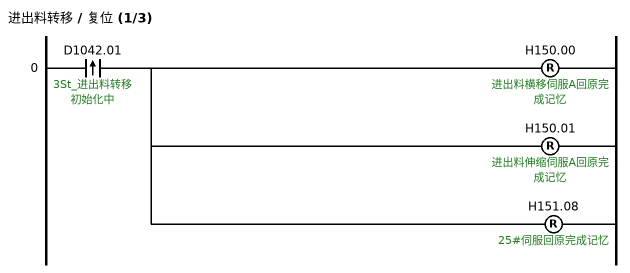
; rung 0
@LD D1042.01  ; 3St_进出料转移 初始化中
RSET H150.00  ; 进出料横移伺服A回原完成记忆
RSET H150.01  ; 进出料伸缩伺服A回原完成记忆
RSET H151.08  ; 25#伺服回原完成记忆

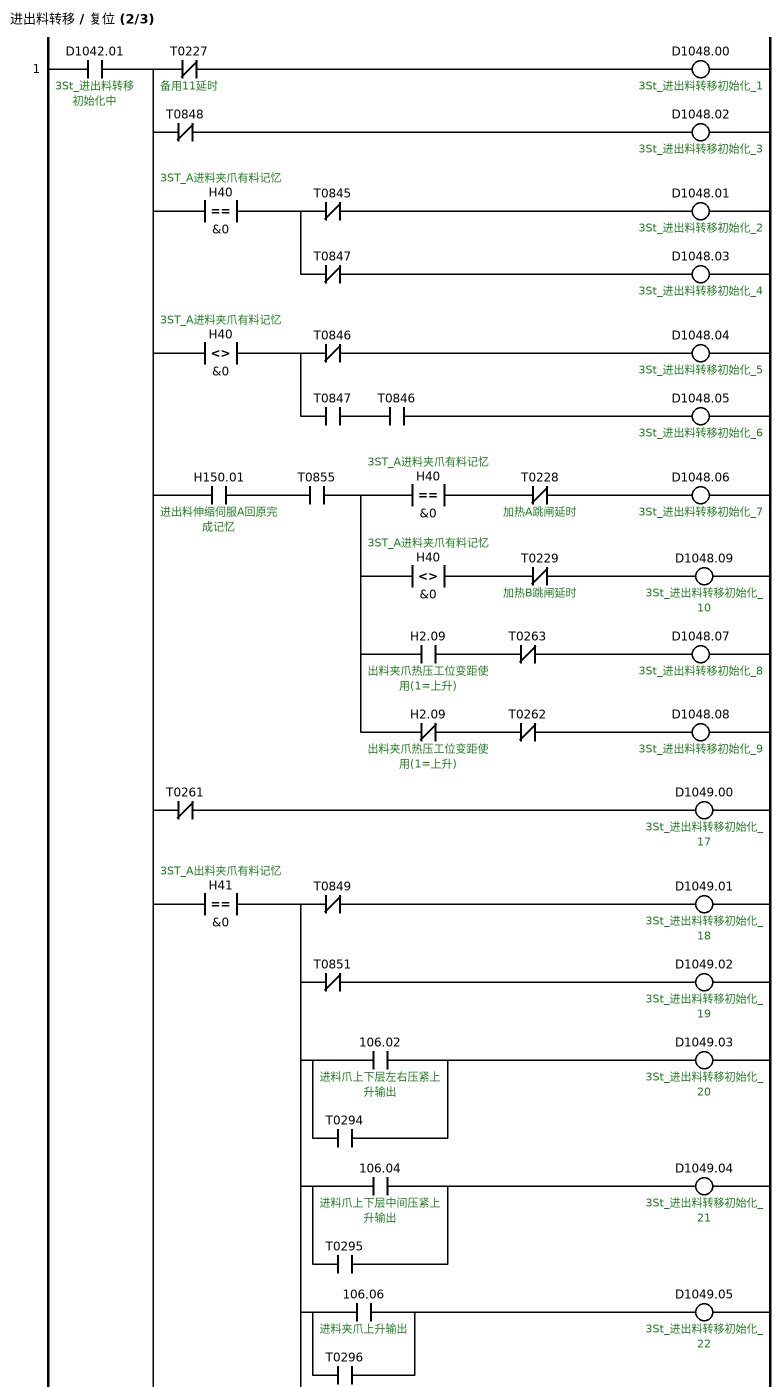

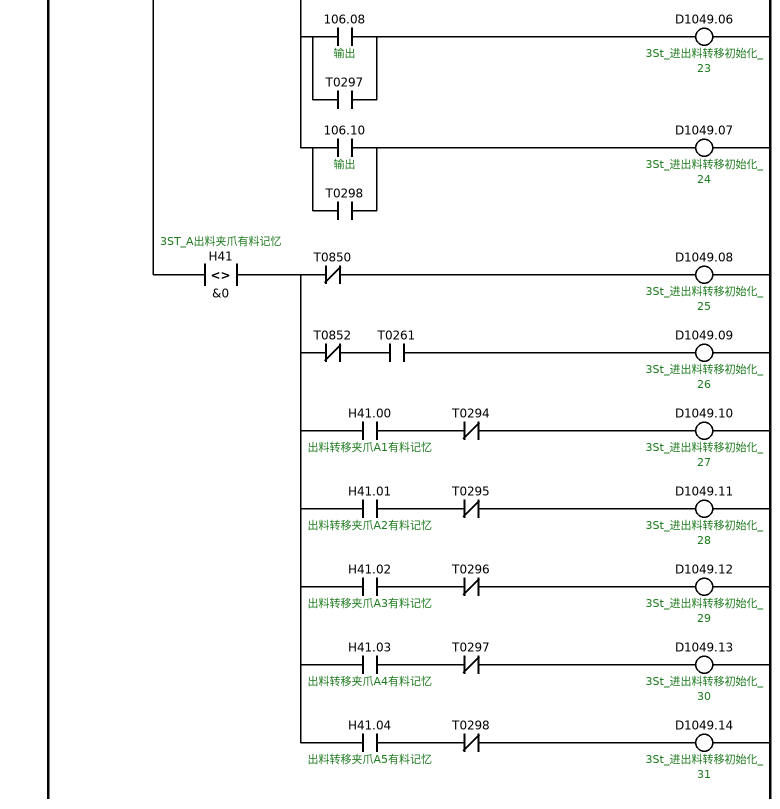
; rung 1
LD D1042.01  ; 3St_进出料转移 初始化中
OUT TR0
ANDNOT T0227  ; 备用11延时
OUT D1048.00  ; 3St_进出料转移初始化_1
LD TR0
ANDNOT T0848
OUT D1048.02  ; 3St_进出料转移初始化_3
LD TR0
AND=(300) H40 &0  ; 3ST_A进料夹爪有料记忆
OUT TR1
ANDNOT T0845
OUT D1048.01  ; 3St_进出料转移初始化_2
LD TR1
ANDNOT T0847
OUT D1048.03  ; 3St_进出料转移初始化_4
LD TR0
AND<>(305) H40 &0  ; 3ST_A进料夹爪有料记忆
OUT TR1
ANDNOT T0846
OUT D1048.04  ; 3St_进出料转移初始化_5
LD TR1
AND T0847
AND T0846
OUT D1048.05  ; 3St_进出料转移初始化_6
LD TR0
AND H150.01  ; 进出料伸缩伺服A回原完成记忆
AND T0855
OUT TR1
AND=(300) H40 &0  ; 3ST_A进料夹爪有料记忆
ANDNOT T0228  ; 加热A跳闸延时
OUT D1048.06  ; 3St_进出料转移初始化_7
LD TR1
AND<>(305) H40 &0  ; 3ST_A进料夹爪有料记忆
ANDNOT T0229  ; 加热B跳闸延时
OUT D1048.09  ; 3St_进出料转移初始化_10
LD TR1
AND H2.09  ; 出料夹爪热压工位变距使用(1=上升)
ANDNOT T0263
OUT D1048.07  ; 3St_进出料转移初始化_8
LD TR1
ANDNOT H2.09  ; 出料夹爪热压工位变距使用(1=上升)
ANDNOT T0262
OUT D1048.08  ; 3St_进出料转移初始化_9
LD TR0
ANDNOT T0261
OUT D1049.00  ; 3St_进出料转移初始化_17
LD TR0
AND=(300) H41 &0  ; 3ST_A出料夹爪有料记忆
OUT TR1
ANDNOT T0849
OUT D1049.01  ; 3St_进出料转移初始化_18
LD TR1
ANDNOT T0851
OUT D1049.02  ; 3St_进出料转移初始化_19
LD TR1
LD 106.02  ; 进料爪上下层左右压紧上升输出
OR T0294
ANDLD
OUT D1049.03  ; 3St_进出料转移初始化_20
LD TR1
LD 106.04  ; 进料爪上下层中间压紧上升输出
OR T0295
ANDLD
OUT D1049.04  ; 3St_进出料转移初始化_21
LD TR1
LD 106.06  ; 进料夹爪上升输出
OR T0296
ANDLD
OUT D1049.05  ; 3St_进出料转移初始化_22
LD TR1
LD 106.08  ; 输出
OR T0297
ANDLD
OUT D1049.06  ; 3St_进出料转移初始化_23
LD TR1
LD 106.10  ; 输出
OR T0298
ANDLD
OUT D1049.07  ; 3St_进出料转移初始化_24
LD TR0
AND<>(305) H41 &0  ; 3ST_A出料夹爪有料记忆
OUT TR0
ANDNOT T0850
OUT D1049.08  ; 3St_进出料转移初始化_25
LD TR0
ANDNOT T0852
AND T0261
OUT D1049.09  ; 3St_进出料转移初始化_26
LD TR0
AND H41.00  ; 出料转移夹爪A1有料记忆
ANDNOT T0294
OUT D1049.10  ; 3St_进出料转移初始化_27
LD TR0
AND H41.01  ; 出料转移夹爪A2有料记忆
ANDNOT T0295
OUT D1049.11  ; 3St_进出料转移初始化_28
LD TR0
AND H41.02  ; 出料转移夹爪A3有料记忆
ANDNOT T0296
OUT D1049.12  ; 3St_进出料转移初始化_29
LD TR0
AND H41.03  ; 出料转移夹爪A4有料记忆
ANDNOT T0297
OUT D1049.13  ; 3St_进出料转移初始化_30
LD TR0
AND H41.04  ; 出料转移夹爪A5有料记忆
ANDNOT T0298
OUT D1049.14  ; 3St_进出料转移初始化_31

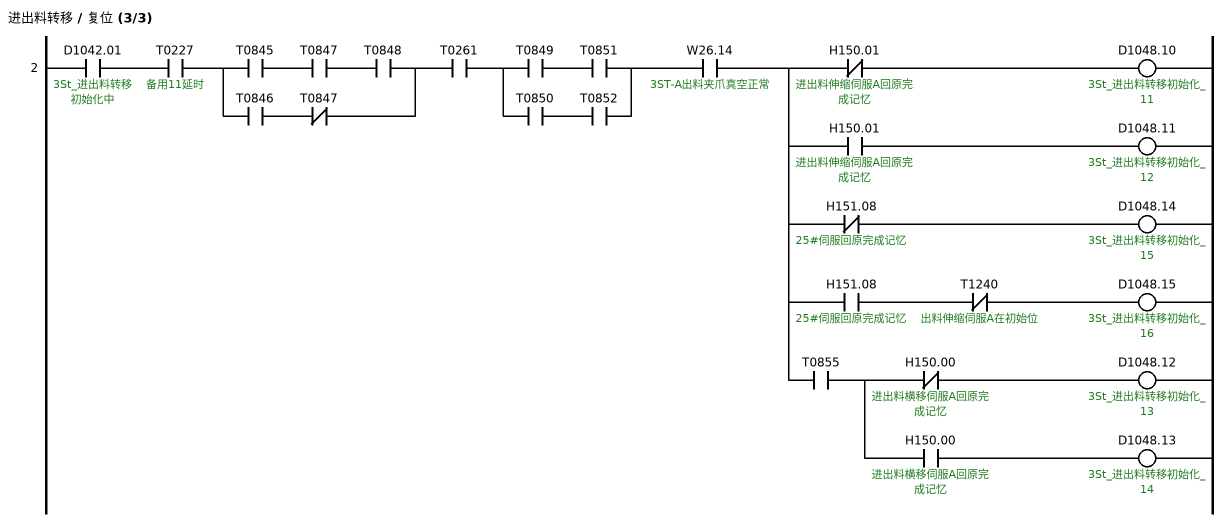
; rung 2
LD D1042.01  ; 3St_进出料转移 初始化中
AND T0227  ; 备用11延时
LD T0845
AND T0847
AND T0848
LD T0846
ANDNOT T0847
ORLD
ANDLD
AND T0261
LD T0849
AND T0851
LD T0850
AND T0852
ORLD
ANDLD
AND W26.14  ; 3ST-A出料夹爪真空正常
OUT TR0
ANDNOT H150.01  ; 进出料伸缩伺服A回原完成记忆
OUT D1048.10  ; 3St_进出料转移初始化_11
LD TR0
AND H150.01  ; 进出料伸缩伺服A回原完成记忆
OUT D1048.11  ; 3St_进出料转移初始化_12
LD TR0
ANDNOT H151.08  ; 25#伺服回原完成记忆
OUT D1048.14  ; 3St_进出料转移初始化_15
LD TR0
AND H151.08  ; 25#伺服回原完成记忆
ANDNOT T1240  ; 出料伸缩伺服A在初始位
OUT D1048.15  ; 3St_进出料转移初始化_16
LD TR0
AND T0855
OUT TR0
ANDNOT H150.00  ; 进出料横移伺服A回原完成记忆
OUT D1048.12  ; 3St_进出料转移初始化_13
LD TR0
AND H150.00  ; 进出料横移伺服A回原完成记忆
OUT D1048.13  ; 3St_进出料转移初始化_14

### Section 输出

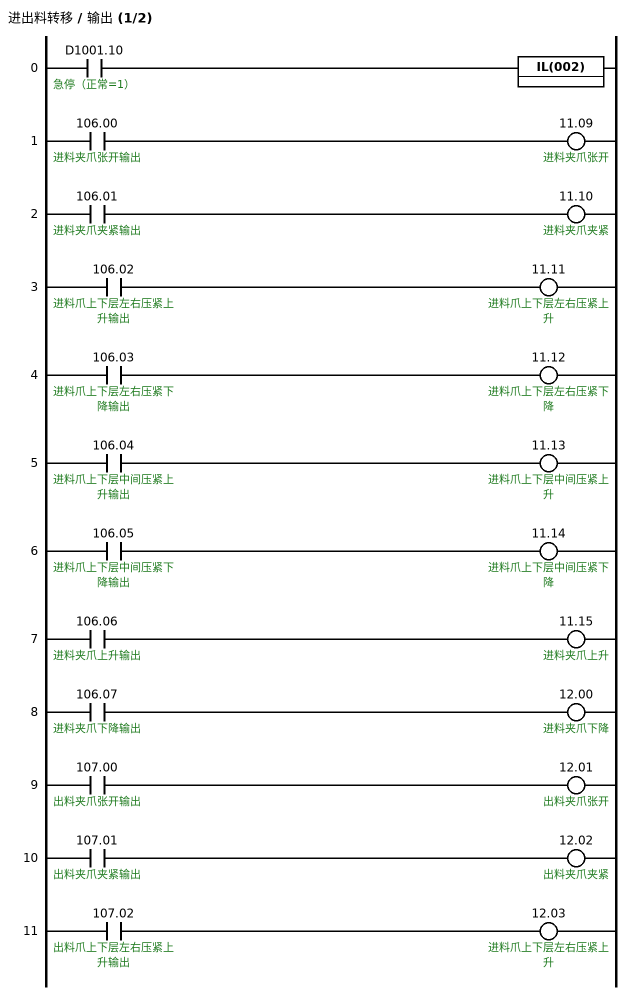
; rung 0
LD D1001.10  ; 急停（正常=1）
IL(002)
; rung 1
LD 106.00  ; 进料夹爪张开输出
OUT 11.09  ; 进料夹爪张开
; rung 2
LD 106.01  ; 进料夹爪夹紧输出
OUT 11.10  ; 进料夹爪夹紧
; rung 3
LD 106.02  ; 进料爪上下层左右压紧上升输出
OUT 11.11  ; 进料爪上下层左右压紧上升
; rung 4
LD 106.03  ; 进料爪上下层左右压紧下降输出
OUT 11.12  ; 进料爪上下层左右压紧下降
; rung 5
LD 106.04  ; 进料爪上下层中间压紧上升输出
OUT 11.13  ; 进料爪上下层中间压紧上升
; rung 6
LD 106.05  ; 进料爪上下层中间压紧下降输出
OUT 11.14  ; 进料爪上下层中间压紧下降
; rung 7
LD 106.06  ; 进料夹爪上升输出
OUT 11.15  ; 进料夹爪上升
; rung 8
LD 106.07  ; 进料夹爪下降输出
OUT 12.00  ; 进料夹爪下降
; rung 9
LD 107.00  ; 出料夹爪张开输出
OUT 12.01  ; 出料夹爪张开
; rung 10
LD 107.01  ; 出料夹爪夹紧输出
OUT 12.02  ; 出料夹爪夹紧
; rung 11
LD 107.02  ; 出料爪上下层左右压紧上升输出
OUT 12.03  ; 进料爪上下层左右压紧上升

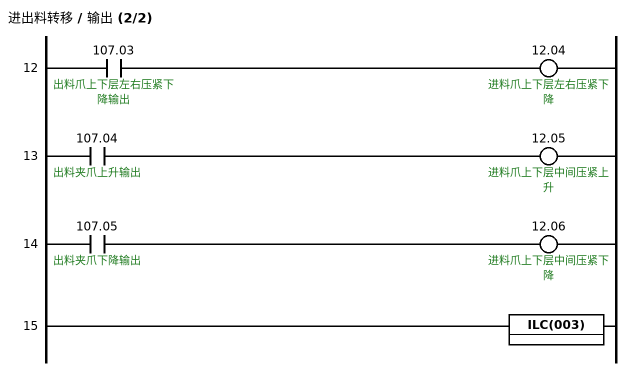
; rung 12
LD 107.03  ; 出料爪上下层左右压紧下降输出
OUT 12.04  ; 进料爪上下层左右压紧下降
; rung 13
LD 107.04  ; 出料夹爪上升输出
OUT 12.05  ; 进料爪上下层中间压紧上升
; rung 14
LD 107.05  ; 出料夹爪下降输出
OUT 12.06  ; 进料爪上下层中间压紧下降
; rung 15
ILC(003)

### Section END
; rung 0
END(001)

## Program 热压A (cyclic task 4)

### Section Main

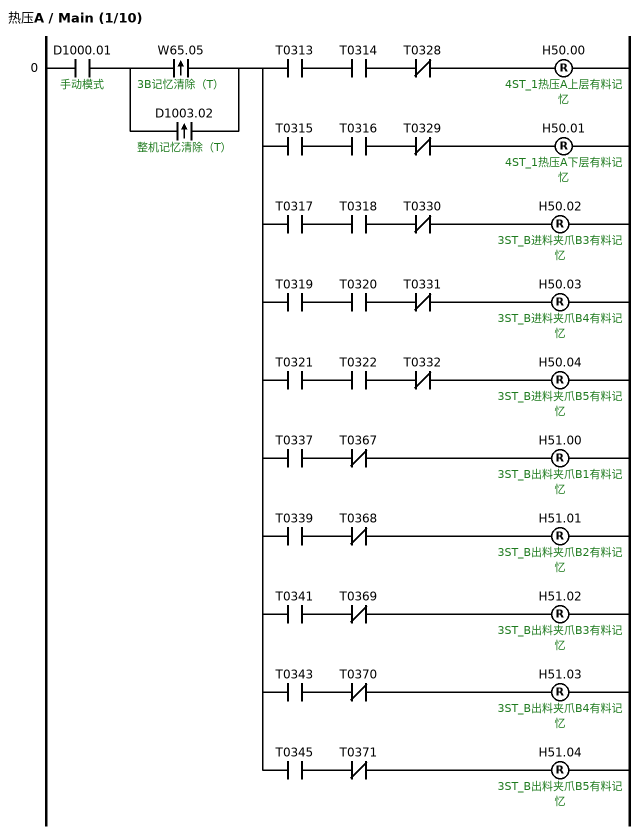
; rung 0
LD D1000.01  ; 手动模式
@LD W65.05  ; 3B记忆清除（T）
@OR D1003.02  ; 整机记忆清除（T）
ANDLD
OUT TR0
AND T0313
AND T0314
ANDNOT T0328
RSET H50.00  ; 4ST_1热压A上层有料记忆
LD TR0
AND T0315
AND T0316
ANDNOT T0329
RSET H50.01  ; 4ST_1热压A下层有料记忆
LD TR0
AND T0317
AND T0318
ANDNOT T0330
RSET H50.02  ; 3ST_B进料夹爪B3有料记忆
LD TR0
AND T0319
AND T0320
ANDNOT T0331
RSET H50.03  ; 3ST_B进料夹爪B4有料记忆
LD TR0
AND T0321
AND T0322
ANDNOT T0332
RSET H50.04  ; 3ST_B进料夹爪B5有料记忆
LD TR0
AND T0337
ANDNOT T0367
RSET H51.00  ; 3ST_B出料夹爪B1有料记忆
LD TR0
AND T0339
ANDNOT T0368
RSET H51.01  ; 3ST_B出料夹爪B2有料记忆
LD TR0
AND T0341
ANDNOT T0369
RSET H51.02  ; 3ST_B出料夹爪B3有料记忆
LD TR0
AND T0343
ANDNOT T0370
RSET H51.03  ; 3ST_B出料夹爪B4有料记忆
LD TR0
AND T0345
ANDNOT T0371
RSET H51.04  ; 3ST_B出料夹爪B5有料记忆

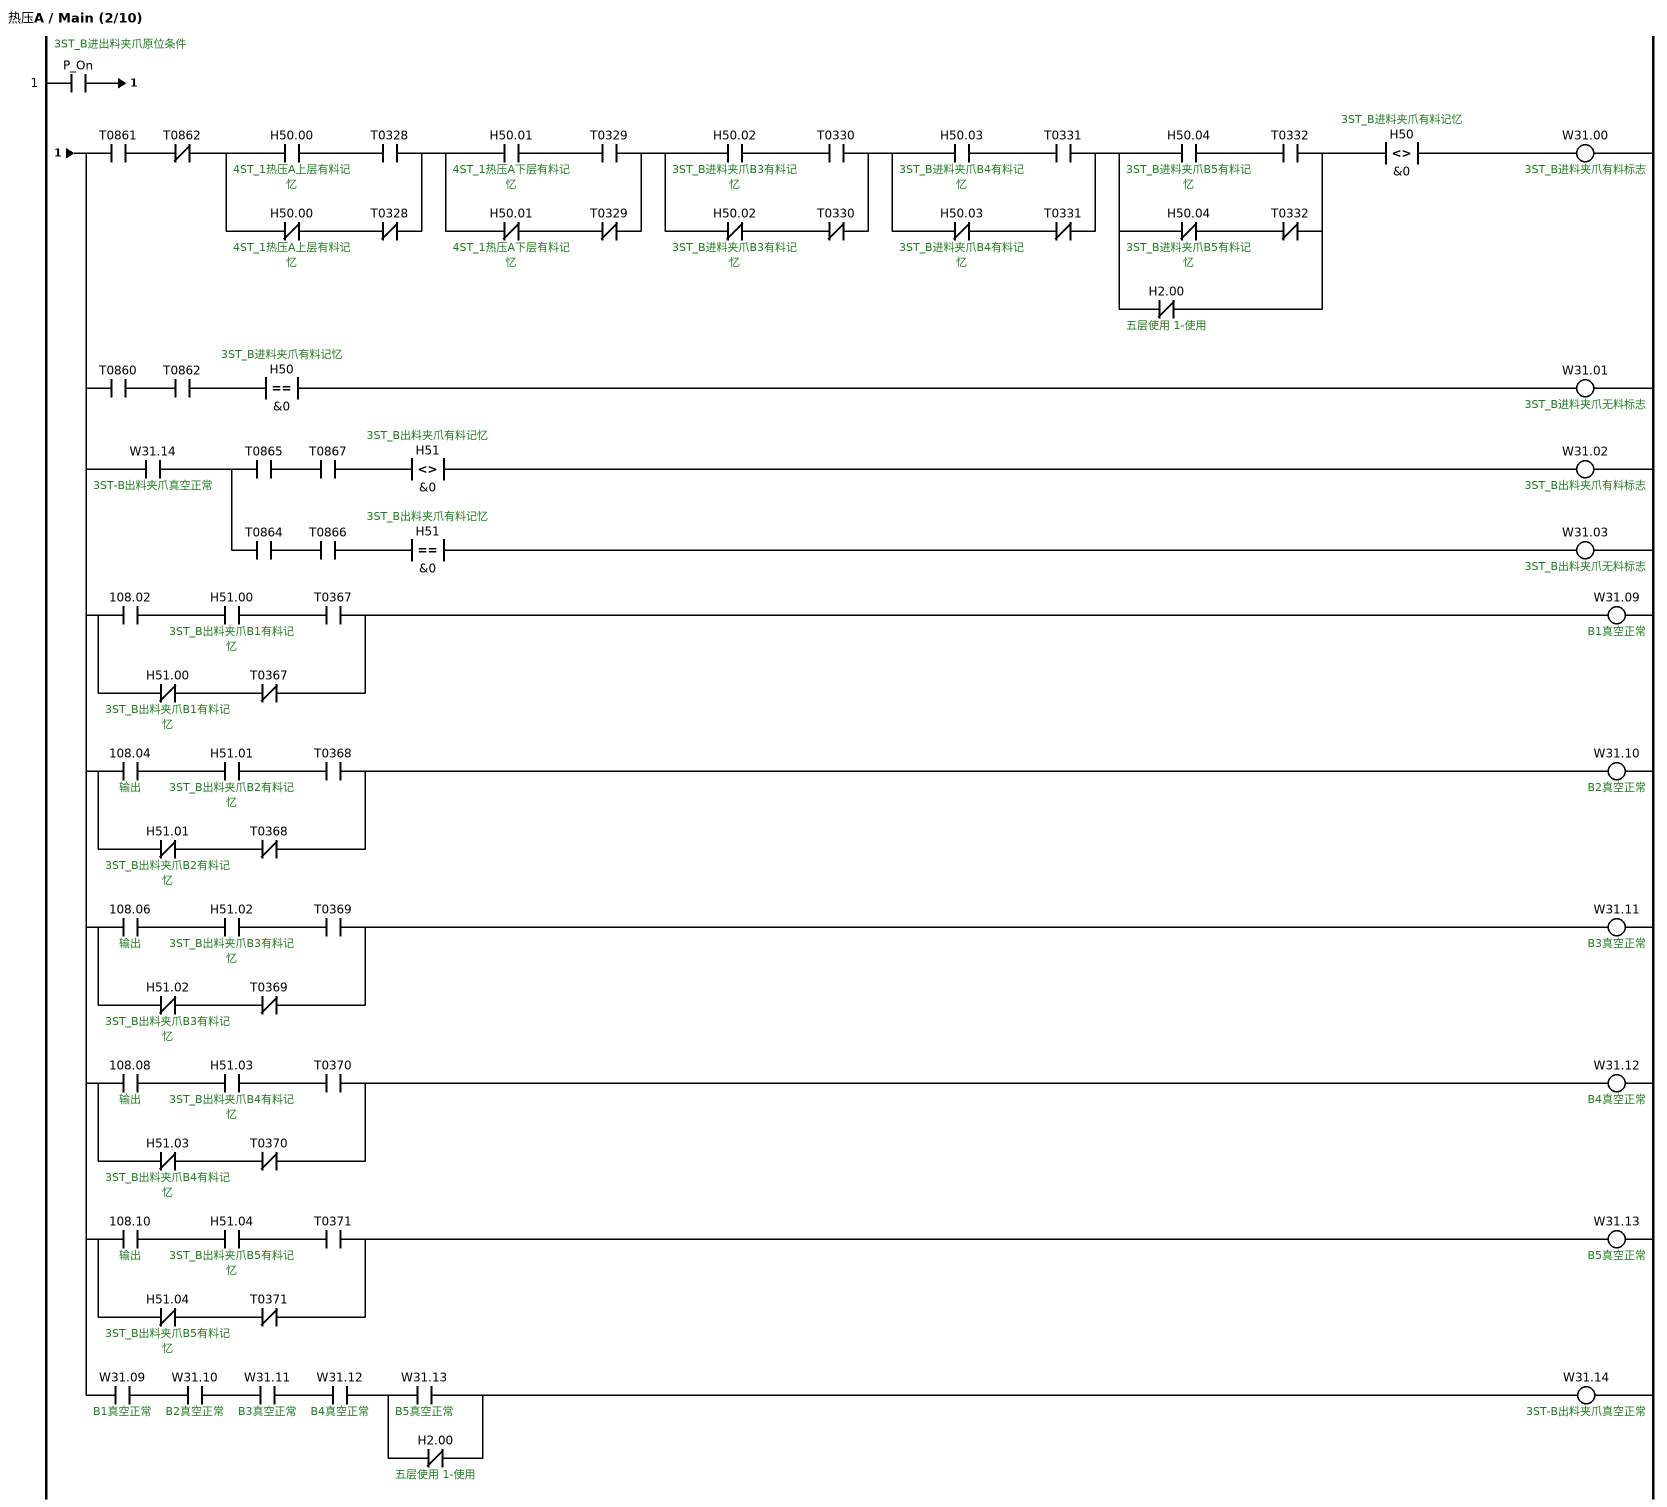
; rung 1: 3ST_B进出料夹爪原位条件
LD P_On
OUT TR0
AND T0861
ANDNOT T0862
LD H50.00  ; 4ST_1热压A上层有料记忆
AND T0328
LDNOT H50.00  ; 4ST_1热压A上层有料记忆
ANDNOT T0328
ORLD
ANDLD
LD H50.01  ; 4ST_1热压A下层有料记忆
AND T0329
LDNOT H50.01  ; 4ST_1热压A下层有料记忆
ANDNOT T0329
ORLD
ANDLD
LD H50.02  ; 3ST_B进料夹爪B3有料记忆
AND T0330
LDNOT H50.02  ; 3ST_B进料夹爪B3有料记忆
ANDNOT T0330
ORLD
ANDLD
LD H50.03  ; 3ST_B进料夹爪B4有料记忆
AND T0331
LDNOT H50.03  ; 3ST_B进料夹爪B4有料记忆
ANDNOT T0331
ORLD
ANDLD
LD H50.04  ; 3ST_B进料夹爪B5有料记忆
AND T0332
LDNOT H50.04  ; 3ST_B进料夹爪B5有料记忆
ANDNOT T0332
ORLD
ORNOT H2.00  ; 五层使用 1-使用
ANDLD
AND<>(305) H50 &0  ; 3ST_B进料夹爪有料记忆
OUT W31.00  ; 3ST_B进料夹爪有料标志
LD TR0
AND T0860
AND T0862
AND=(300) H50 &0  ; 3ST_B进料夹爪有料记忆
OUT W31.01  ; 3ST_B进料夹爪无料标志
LD TR0
AND W31.14  ; 3ST-B出料夹爪真空正常
OUT TR1
AND T0865
AND T0867
AND<>(305) H51 &0  ; 3ST_B出料夹爪有料记忆
OUT W31.02  ; 3ST_B出料夹爪有料标志
LD TR1
AND T0864
AND T0866
AND=(300) H51 &0  ; 3ST_B出料夹爪有料记忆
OUT W31.03  ; 3ST_B出料夹爪无料标志
LD TR0
LD 108.02
AND H51.00  ; 3ST_B出料夹爪B1有料记忆
AND T0367
LDNOT H51.00  ; 3ST_B出料夹爪B1有料记忆
ANDNOT T0367
ORLD
ANDLD
OUT W31.09  ; B1真空正常
LD TR0
LD 108.04  ; 输出
AND H51.01  ; 3ST_B出料夹爪B2有料记忆
AND T0368
LDNOT H51.01  ; 3ST_B出料夹爪B2有料记忆
ANDNOT T0368
ORLD
ANDLD
OUT W31.10  ; B2真空正常
LD TR0
LD 108.06  ; 输出
AND H51.02  ; 3ST_B出料夹爪B3有料记忆
AND T0369
LDNOT H51.02  ; 3ST_B出料夹爪B3有料记忆
ANDNOT T0369
ORLD
ANDLD
OUT W31.11  ; B3真空正常
LD TR0
LD 108.08  ; 输出
AND H51.03  ; 3ST_B出料夹爪B4有料记忆
AND T0370
LDNOT H51.03  ; 3ST_B出料夹爪B4有料记忆
ANDNOT T0370
ORLD
ANDLD
OUT W31.12  ; B4真空正常
LD TR0
LD 108.10  ; 输出
AND H51.04  ; 3ST_B出料夹爪B5有料记忆
AND T0371
LDNOT H51.04  ; 3ST_B出料夹爪B5有料记忆
ANDNOT T0371
ORLD
ANDLD
OUT W31.13  ; B5真空正常
LD TR0
AND W31.09  ; B1真空正常
AND W31.10  ; B2真空正常
AND W31.11  ; B3真空正常
AND W31.12  ; B4真空正常
LD W31.13  ; B5真空正常
ORNOT H2.00  ; 五层使用 1-使用
ANDLD
OUT W31.14  ; 3ST-B出料夹爪真空正常

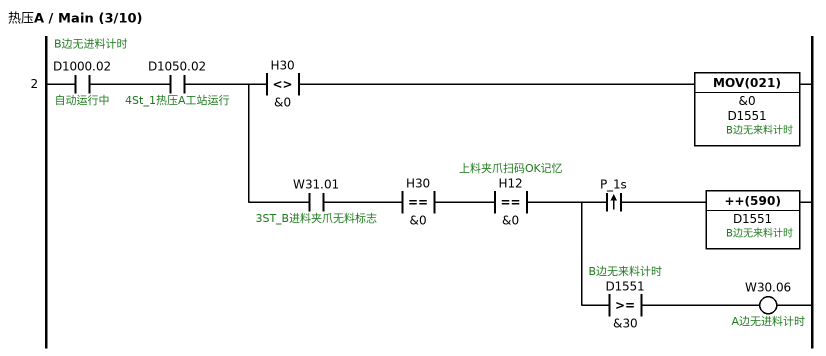
; rung 2: B边无进料计时
LD D1000.02  ; 自动运行中
AND D1050.02  ; 4St_1热压A工站运行
OUT TR0
AND<>(305) H30 &0
MOV(021) &0 D1551  ; B边无来料计时
LD TR0
AND W31.01  ; 3ST_B进料夹爪无料标志
AND=(300) H30 &0
AND=(300) H12 &0  ; 上料夹爪扫码OK记忆
OUT TR0
@AND P_1s
++(590) D1551  ; B边无来料计时
LD TR0
AND>=(325) D1551 &30  ; B边无来料计时
OUT W30.06  ; A边无进料计时

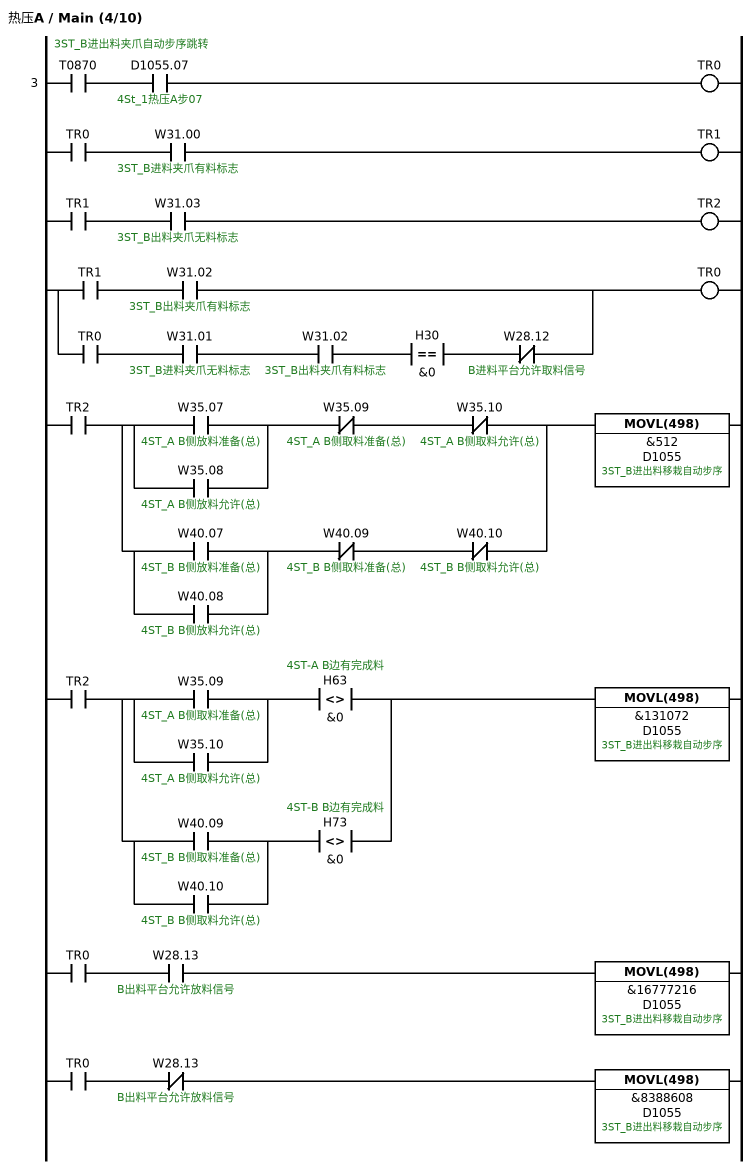
; rung 3: 3ST_B进出料夹爪自动步序跳转
LD T0870
AND D1055.07  ; 4St_1热压A步07
OUT TR0
AND W31.00  ; 3ST_B进料夹爪有料标志
OUT TR1
AND W31.03  ; 3ST_B出料夹爪无料标志
OUT TR2
LD W35.07  ; 4ST_A B侧放料准备(总)
OR W35.08  ; 4ST_A B侧放料允许(总)
ANDNOT W35.09  ; 4ST_A B侧取料准备(总)
ANDNOT W35.10  ; 4ST_A B侧取料允许(总)
LD W40.07  ; 4ST_B B侧放料准备(总)
OR W40.08  ; 4ST_B B侧放料允许(总)
ANDNOT W40.09  ; 4ST_B B侧取料准备(总)
ANDNOT W40.10  ; 4ST_B B侧取料允许(总)
ORLD
ANDLD
MOVL(498) &512 D1055  ; 3ST_B进出料移栽自动步序  // D1055.09  3ST_B到热压上料位
LD TR2
LD W35.09  ; 4ST_A B侧取料准备(总)
OR W35.10  ; 4ST_A B侧取料允许(总)
AND<>(305) H63 &0  ; 4ST-A B边有完成料
LD W40.09  ; 4ST_B B侧取料准备(总)
OR W40.10  ; 4ST_B B侧取料允许(总)
AND<>(305) H73 &0  ; 4ST-B B边有完成料
ORLD
ANDLD
MOVL(498) &131072 D1055  ; 3ST_B进出料移栽自动步序  // D1056.01  3ST_B到热压下料位
LD TR1
AND W31.02  ; 3ST_B出料夹爪有料标志
LD TR0
AND W31.01  ; 3ST_B进料夹爪无料标志
AND W31.02  ; 3ST_B出料夹爪有料标志
AND=(300) H30 &0
ANDNOT W28.12  ; B进料平台允许取料信号
ORLD
OUT TR0
AND W28.13  ; B出料平台允许放料信号
MOVL(498) &16777216 D1055  ; 3ST_B进出料移栽自动步序  // D1056.08  3ST_B到出料位出料/夹爪下降
LD TR0
ANDNOT W28.13  ; B出料平台允许放料信号
MOVL(498) &8388608 D1055  ; 3ST_B进出料移栽自动步序  // D1056.07  3ST_B到出料等待位

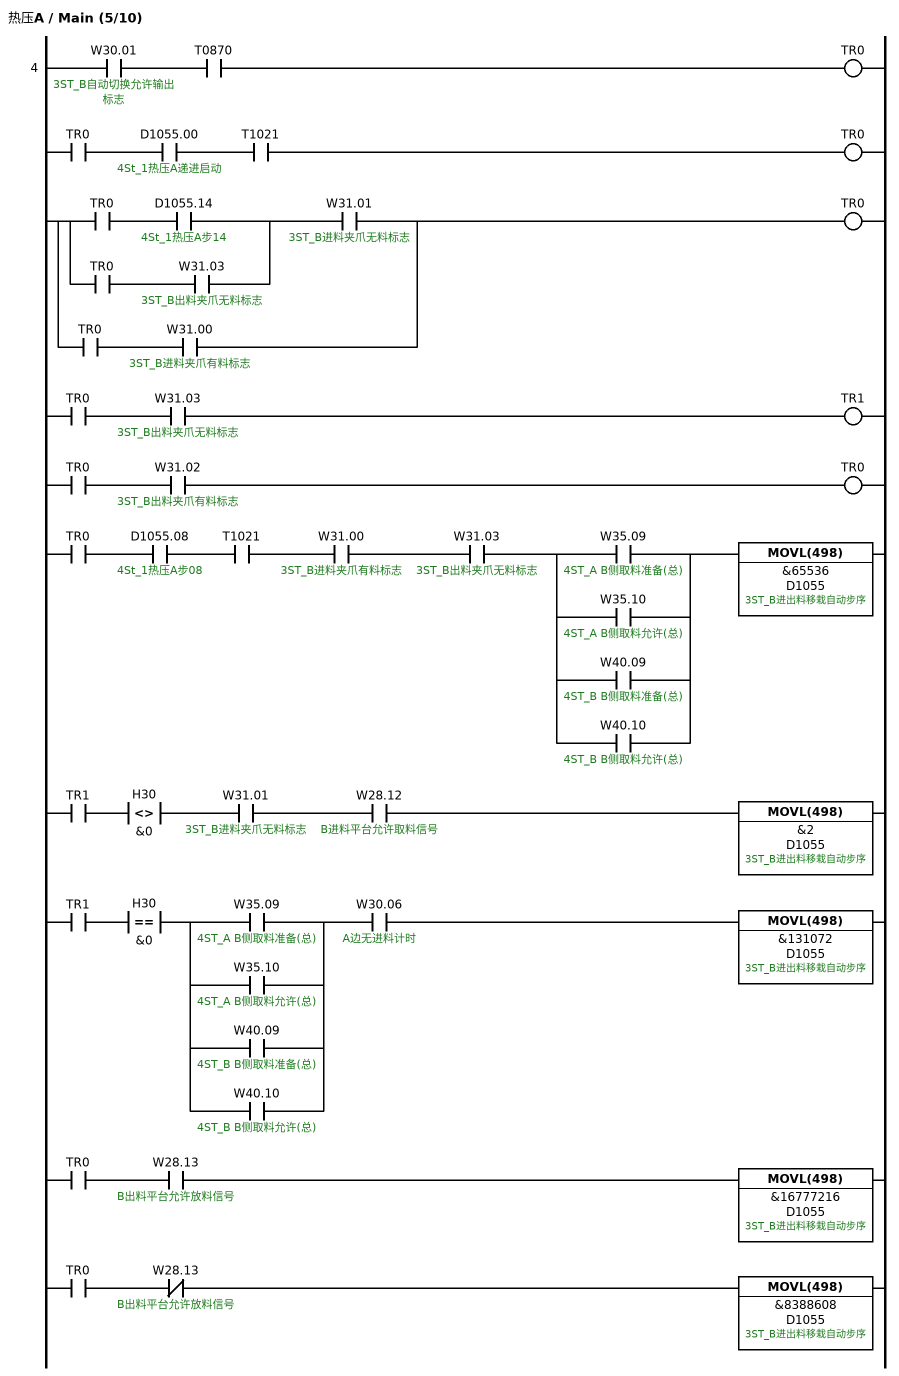
; rung 4
LD W30.01  ; 3ST_B自动切换允许输出标志
AND T0870
OUT TR0
AND D1055.08  ; 4St_1热压A步08
AND T1021
AND W31.00  ; 3ST_B进料夹爪有料标志
AND W31.03  ; 3ST_B出料夹爪无料标志
LD W35.09  ; 4ST_A B侧取料准备(总)
OR W35.10  ; 4ST_A B侧取料允许(总)
OR W40.09  ; 4ST_B B侧取料准备(总)
OR W40.10  ; 4ST_B B侧取料允许(总)
ANDLD
MOVL(498) &65536 D1055  ; 3ST_B进出料移栽自动步序  // D1056.01  3ST_B热压工位下料需求
LD TR0
AND D1055.14  ; 4St_1热压A步14
LD TR0
AND D1055.00  ; 4St_1热压A递进启动
AND T1021
OUT TR0
AND W31.03  ; 3ST_B出料夹爪无料标志
ORLD
AND W31.01  ; 3ST_B进料夹爪无料标志
LD TR0
AND W31.00  ; 3ST_B进料夹爪有料标志
ORLD
OUT TR0
AND W31.03  ; 3ST_B出料夹爪无料标志
OUT TR1
AND<>(305) H30 &0
AND W31.01  ; 3ST_B进料夹爪无料标志
AND W28.12  ; B进料平台允许取料信号
MOVL(498) &2 D1055  ; 3ST_B进出料移栽自动步序  // D1055.02  3ST_B到进料位
LD TR1
AND=(300) H30 &0
LD W35.09  ; 4ST_A B侧取料准备(总)
OR W35.10  ; 4ST_A B侧取料允许(总)
OR W40.09  ; 4ST_B B侧取料准备(总)
OR W40.10  ; 4ST_B B侧取料允许(总)
ANDLD
AND W30.06  ; A边无进料计时
MOVL(498) &131072 D1055  ; 3ST_B进出料移栽自动步序  // D1056.01  3ST_B到热压下料位
LD TR0
AND W31.02  ; 3ST_B出料夹爪有料标志
OUT TR0
AND W28.13  ; B出料平台允许放料信号
MOVL(498) &16777216 D1055  ; 3ST_B进出料移栽自动步序  // D1056.08  3ST_B到出料位出料/夹爪下降
LD TR0
ANDNOT W28.13  ; B出料平台允许放料信号
MOVL(498) &8388608 D1055  ; 3ST_B进出料移栽自动步序  // D1056.07  3ST_B到出料等待位

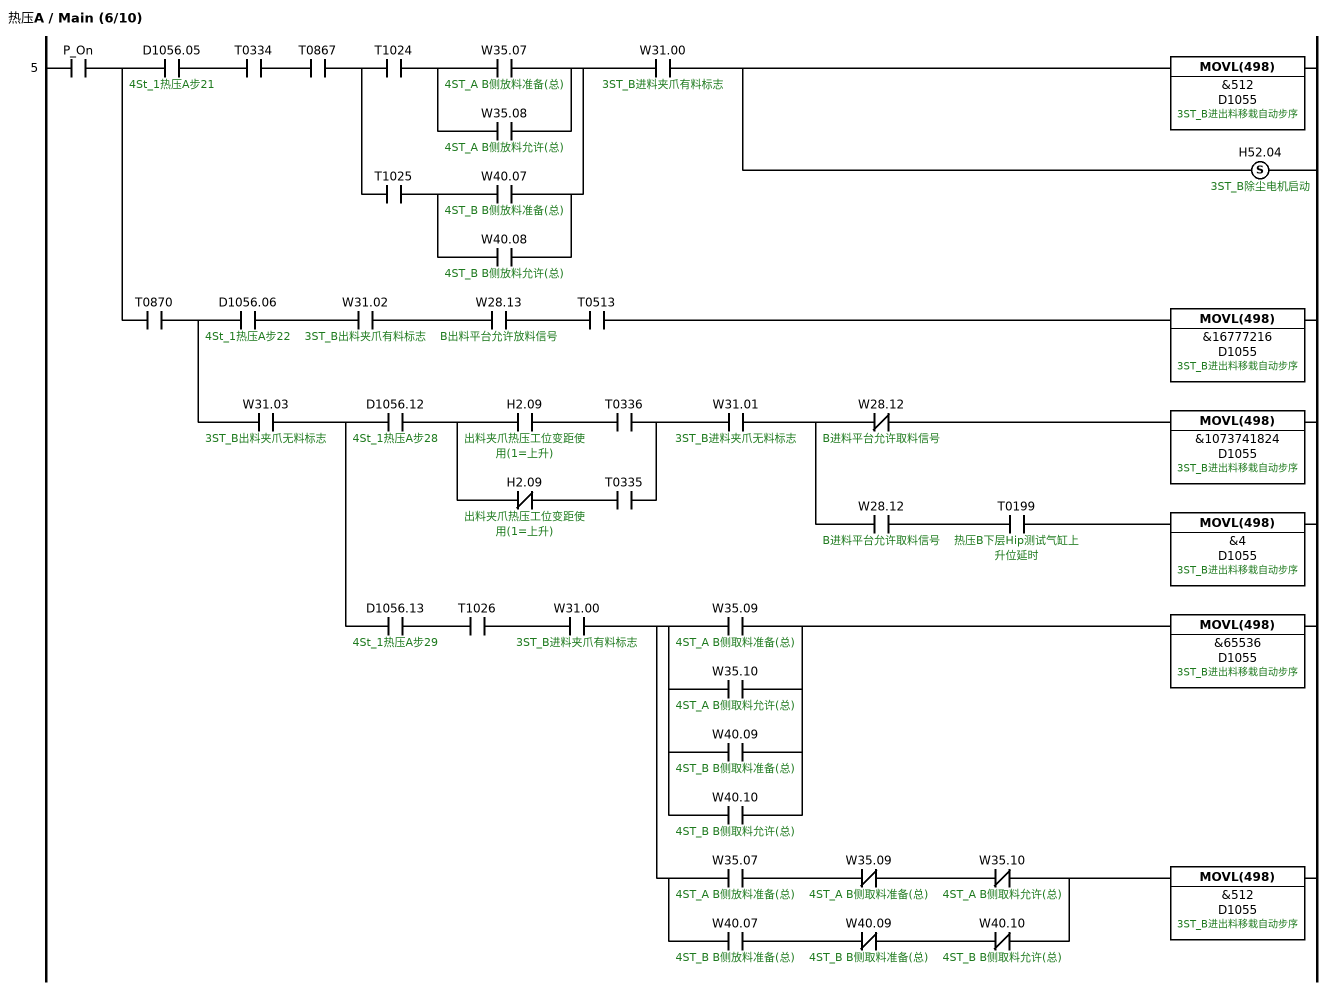
; rung 5
LD P_On
OUT TR0
AND D1056.05  ; 4St_1热压A步21
AND T0334
AND T0867
LD T1024
LD W35.07  ; 4ST_A B侧放料准备(总)
OR W35.08  ; 4ST_A B侧放料允许(总)
ANDLD
LD T1025
LD W40.07  ; 4ST_B B侧放料准备(总)
OR W40.08  ; 4ST_B B侧放料允许(总)
ANDLD
ORLD
ANDLD
AND W31.00  ; 3ST_B进料夹爪有料标志
MOVL(498) &512 D1055  ; 3ST_B进出料移栽自动步序  // D1055.09  3ST_B到热压上料位
SET H52.04  ; 3ST_B除尘电机启动
LD TR0
AND T0870
OUT TR0
AND D1056.06  ; 4St_1热压A步22
AND W31.02  ; 3ST_B出料夹爪有料标志
AND W28.13  ; B出料平台允许放料信号
AND T0513
MOVL(498) &16777216 D1055  ; 3ST_B进出料移栽自动步序  // D1056.08  3ST_B到出料位出料
LD TR0
AND W31.03  ; 3ST_B出料夹爪无料标志
OUT TR0
AND D1056.12  ; 4St_1热压A步28
LD H2.09  ; 出料夹爪热压工位变距使用(1=上升)
AND T0336
LDNOT H2.09  ; 出料夹爪热压工位变距使用(1=上升)
AND T0335
ORLD
ANDLD
AND W31.01  ; 3ST_B进料夹爪无料标志
OUT TR1
ANDNOT W28.12  ; B进料平台允许取料信号
MOVL(498) &1073741824 D1055  ; 3ST_B进出料移栽自动步序  // D1055.14  3ST_B进出料横移伺服到进料等待位
LD TR1
AND W28.12  ; B进料平台允许取料信号
AND T0199  ; 热压B下层Hip测试气缸上升位延时
MOVL(498) &4 D1055  ; 3ST_B进出料移栽自动步序  // D1055.02  3ST_B到进料位
LD TR0
AND D1056.13  ; 4St_1热压A步29
AND T1026
AND W31.00  ; 3ST_B进料夹爪有料标志
OUT TR0
LD W35.09  ; 4ST_A B侧取料准备(总)
OR W35.10  ; 4ST_A B侧取料允许(总)
OR W40.09  ; 4ST_B B侧取料准备(总)
OR W40.10  ; 4ST_B B侧取料允许(总)
ANDLD
MOVL(498) &65536 D1055  ; 3ST_B进出料移栽自动步序  // D1056.00  3ST_B热压工位下料需求
LD TR0
LD W35.07  ; 4ST_A B侧放料准备(总)
ANDNOT W35.09  ; 4ST_A B侧取料准备(总)
ANDNOT W35.10  ; 4ST_A B侧取料允许(总)
LD W40.07  ; 4ST_B B侧放料准备(总)
ANDNOT W40.09  ; 4ST_B B侧取料准备(总)
ANDNOT W40.10  ; 4ST_B B侧取料允许(总)
ORLD
ANDLD
MOVL(498) &512 D1055  ; 3ST_B进出料移栽自动步序  // D1055.09  3ST_B到热压上料位

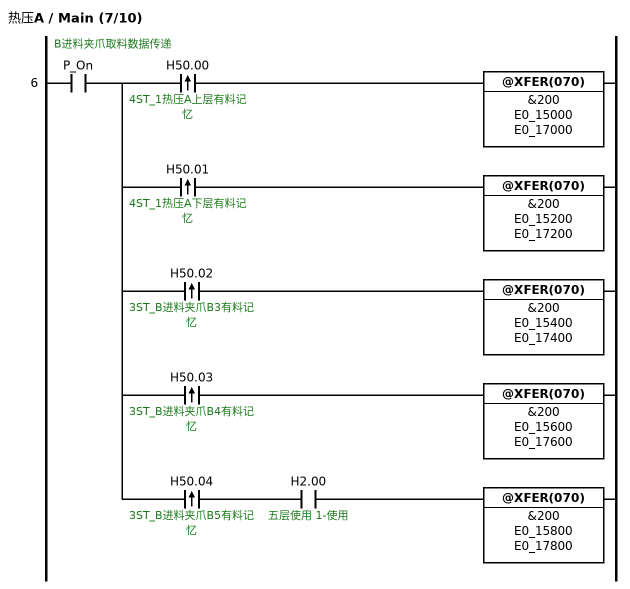
; rung 6: B进料夹爪取料数据传递
LD P_On
OUT TR0
@AND H50.00  ; 4ST_1热压A上层有料记忆
@XFER(070) &200 E0_15000 E0_17000
LD TR0
@AND H50.01  ; 4ST_1热压A下层有料记忆
@XFER(070) &200 E0_15200 E0_17200
LD TR0
@AND H50.02  ; 3ST_B进料夹爪B3有料记忆
@XFER(070) &200 E0_15400 E0_17400
LD TR0
@AND H50.03  ; 3ST_B进料夹爪B4有料记忆
@XFER(070) &200 E0_15600 E0_17600
LD TR0
@AND H50.04  ; 3ST_B进料夹爪B5有料记忆
AND H2.00  ; 五层使用 1-使用
@XFER(070) &200 E0_15800 E0_17800

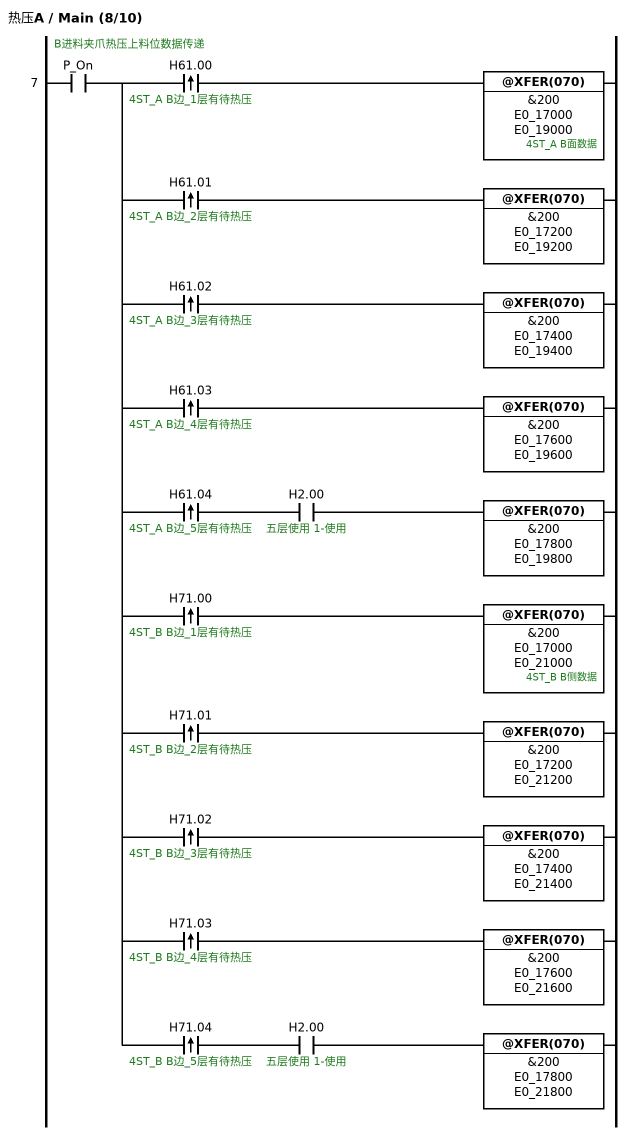
; rung 7: B进料夹爪热压上料位数据传递
LD P_On
OUT TR0
@AND H61.00  ; 4ST_A B边_1层有待热压
@XFER(070) &200 E0_17000 E0_19000  ; 4ST_A B面数据
LD TR0
@AND H61.01  ; 4ST_A B边_2层有待热压
@XFER(070) &200 E0_17200 E0_19200
LD TR0
@AND H61.02  ; 4ST_A B边_3层有待热压
@XFER(070) &200 E0_17400 E0_19400
LD TR0
@AND H61.03  ; 4ST_A B边_4层有待热压
@XFER(070) &200 E0_17600 E0_19600
LD TR0
@AND H61.04  ; 4ST_A B边_5层有待热压
AND H2.00  ; 五层使用 1-使用
@XFER(070) &200 E0_17800 E0_19800
LD TR0
@AND H71.00  ; 4ST_B B边_1层有待热压
@XFER(070) &200 E0_17000 E0_21000  ; 4ST_B B侧数据
LD TR0
@AND H71.01  ; 4ST_B B边_2层有待热压
@XFER(070) &200 E0_17200 E0_21200
LD TR0
@AND H71.02  ; 4ST_B B边_3层有待热压
@XFER(070) &200 E0_17400 E0_21400
LD TR0
@AND H71.03  ; 4ST_B B边_4层有待热压
@XFER(070) &200 E0_17600 E0_21600
LD TR0
@AND H71.04  ; 4ST_B B边_5层有待热压
AND H2.00  ; 五层使用 1-使用
@XFER(070) &200 E0_17800 E0_21800

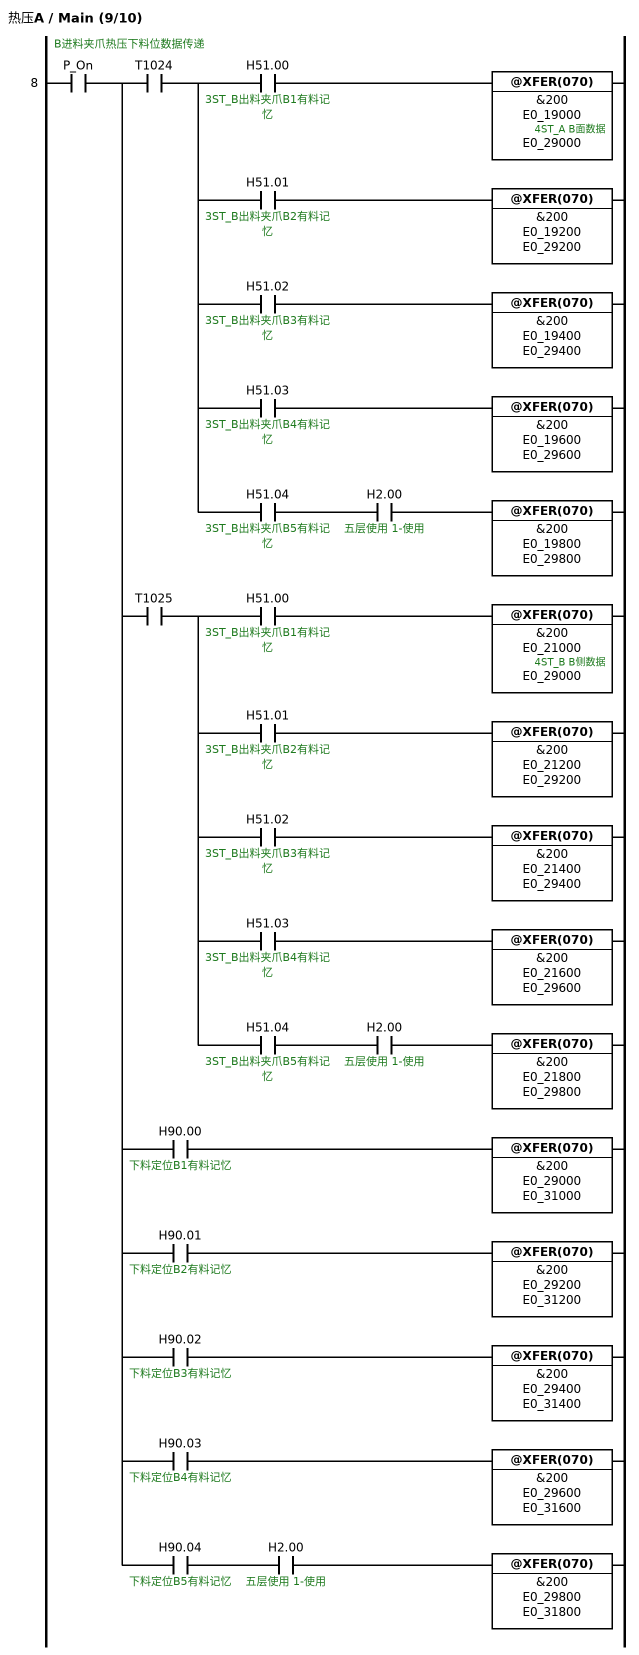
; rung 8: B进料夹爪热压下料位数据传递
LD P_On
OUT TR0
AND T1024
OUT TR1
AND H51.00  ; 3ST_B出料夹爪B1有料记忆
@XFER(070) &200 E0_19000 E0_29000  ; 4ST_A B面数据
LD TR1
AND H51.01  ; 3ST_B出料夹爪B2有料记忆
@XFER(070) &200 E0_19200 E0_29200
LD TR1
AND H51.02  ; 3ST_B出料夹爪B3有料记忆
@XFER(070) &200 E0_19400 E0_29400
LD TR1
AND H51.03  ; 3ST_B出料夹爪B4有料记忆
@XFER(070) &200 E0_19600 E0_29600
LD TR1
AND H51.04  ; 3ST_B出料夹爪B5有料记忆
AND H2.00  ; 五层使用 1-使用
@XFER(070) &200 E0_19800 E0_29800
LD TR0
AND T1025
OUT TR1
AND H51.00  ; 3ST_B出料夹爪B1有料记忆
@XFER(070) &200 E0_21000 E0_29000  ; 4ST_B B侧数据
LD TR1
AND H51.01  ; 3ST_B出料夹爪B2有料记忆
@XFER(070) &200 E0_21200 E0_29200
LD TR1
AND H51.02  ; 3ST_B出料夹爪B3有料记忆
@XFER(070) &200 E0_21400 E0_29400
LD TR1
AND H51.03  ; 3ST_B出料夹爪B4有料记忆
@XFER(070) &200 E0_21600 E0_29600
LD TR1
AND H51.04  ; 3ST_B出料夹爪B5有料记忆
AND H2.00  ; 五层使用 1-使用
@XFER(070) &200 E0_21800 E0_29800
LD TR0
AND H90.00  ; 下料定位B1有料记忆
@XFER(070) &200 E0_29000 E0_31000
LD TR0
AND H90.01  ; 下料定位B2有料记忆
@XFER(070) &200 E0_29200 E0_31200
LD TR0
AND H90.02  ; 下料定位B3有料记忆
@XFER(070) &200 E0_29400 E0_31400
LD TR0
AND H90.03  ; 下料定位B4有料记忆
@XFER(070) &200 E0_29600 E0_31600
LD TR0
AND H90.04  ; 下料定位B5有料记忆
AND H2.00  ; 五层使用 1-使用
@XFER(070) &200 E0_29800 E0_31800

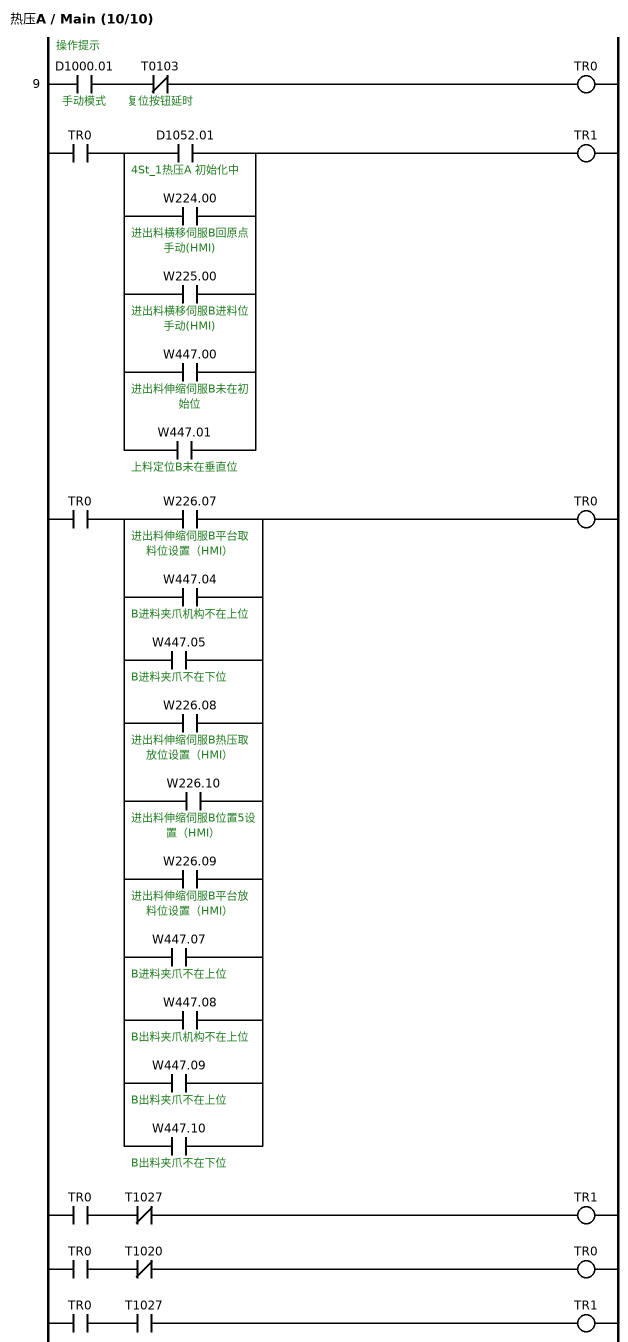

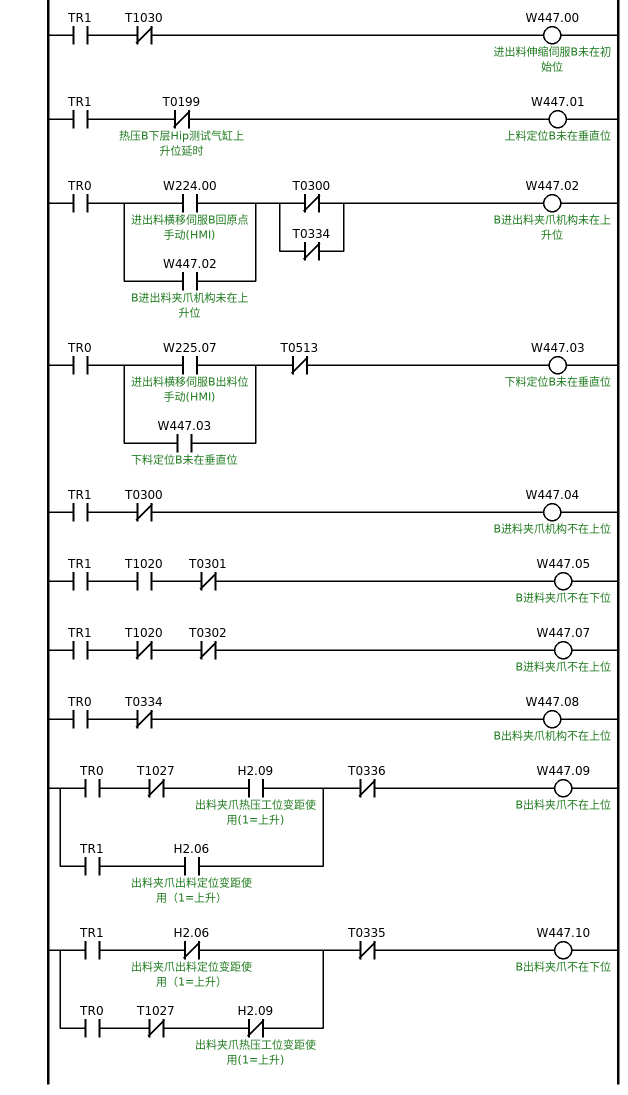
; rung 9: 操作提示
LD D1000.01  ; 手动模式
ANDNOT T0103  ; 复位按钮延时
OUT TR0
LD D1052.01  ; 4St_1热压A 初始化中
OR W224.00  ; 进出料横移伺服B回原点手动(HMI)
OR W225.00  ; 进出料横移伺服B进料位手动(HMI)
OR W447.00  ; 进出料伸缩伺服B未在初始位
OR W447.01  ; 上料定位B未在垂直位
ANDLD
OUT TR1
ANDNOT T1030
OUT W447.00  ; 进出料伸缩伺服B未在初始位
LD TR1
ANDNOT T0199  ; 热压B下层Hip测试气缸上升位延时
OUT W447.01  ; 上料定位B未在垂直位
LD TR0
LD W224.00  ; 进出料横移伺服B回原点手动(HMI)
OR W447.02  ; B进出料夹爪机构未在上升位
ANDLD
LDNOT T0300
ORNOT T0334
ANDLD
OUT W447.02  ; B进出料夹爪机构未在上升位
LD TR0
LD W225.07  ; 进出料横移伺服B出料位手动(HMI)
OR W447.03  ; 下料定位B未在垂直位
ANDLD
ANDNOT T0513
OUT W447.03  ; 下料定位B未在垂直位
LD TR0
LD W226.07  ; 进出料伸缩伺服B平台取料位设置（HMI）
OR W447.04  ; B进料夹爪机构不在上位
OR W447.05  ; B进料夹爪不在下位
OR W226.08  ; 进出料伸缩伺服B热压取放位设置（HMI）
OR W226.10  ; 进出料伸缩伺服B位置5设置（HMI）
OR W226.09  ; 进出料伸缩伺服B平台放料位设置（HMI）
OR W447.07  ; B进料夹爪不在上位
OR W447.08  ; B出料夹爪机构不在上位
OR W447.09  ; B出料夹爪不在上位
OR W447.10  ; B出料夹爪不在下位
ANDLD
OUT TR0
ANDNOT T1027
OUT TR1
ANDNOT T0300
OUT W447.04  ; B进料夹爪机构不在上位
LD TR1
AND T1020
ANDNOT T0301
OUT W447.05  ; B进料夹爪不在下位
LD TR1
ANDNOT T1020
ANDNOT T0302
OUT W447.07  ; B进料夹爪不在上位
LD TR0
ANDNOT T1020
OUT TR0
ANDNOT T0334
OUT W447.08  ; B出料夹爪机构不在上位
LD TR0
ANDNOT T1027
AND H2.09  ; 出料夹爪热压工位变距使用(1=上升)
LD TR0
AND T1027
OUT TR1
AND H2.06  ; 出料夹爪出料定位变距使用（1=上升）
ORLD
ANDNOT T0336
OUT W447.09  ; B出料夹爪不在上位
LD TR1
ANDNOT H2.06  ; 出料夹爪出料定位变距使用（1=上升）
LD TR0
ANDNOT T1027
ANDNOT H2.09  ; 出料夹爪热压工位变距使用(1=上升)
ORLD
ANDNOT T0335
OUT W447.10  ; B出料夹爪不在下位

### Section _4ST_1热压A

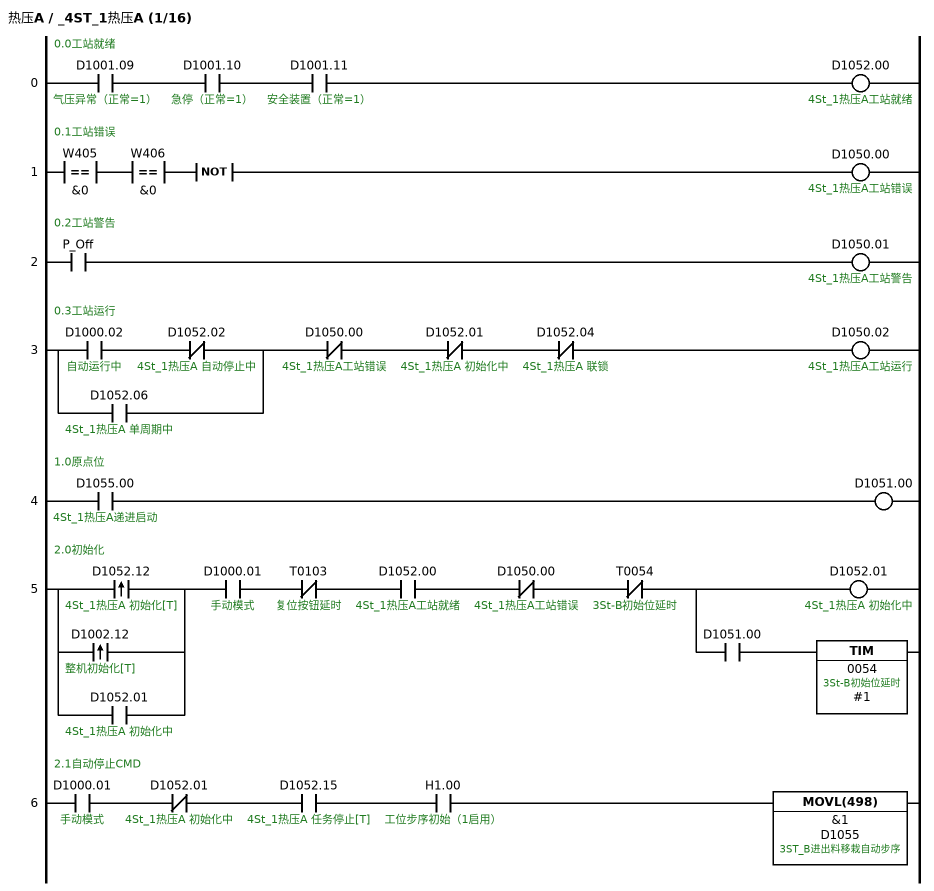
; rung 0: 0.0工站就绪
LD D1001.09  ; 气压异常（正常=1）
AND D1001.10  ; 急停（正常=1）
AND D1001.11  ; 安全装置（正常=1）
OUT D1052.00  ; 4St_1热压A工站就绪
; rung 1: 0.1工站错误
LD=(300) W405 &0
AND=(300) W406 &0
NOT(520)
OUT D1050.00  ; 4St_1热压A工站错误
; rung 2: 0.2工站警告
LD P_Off
OUT D1050.01  ; 4St_1热压A工站警告
; rung 3: 0.3工站运行
LD D1000.02  ; 自动运行中
ANDNOT D1052.02  ; 4St_1热压A 自动停止中
OR D1052.06  ; 4St_1热压A 单周期中
ANDNOT D1050.00  ; 4St_1热压A工站错误
ANDNOT D1052.01  ; 4St_1热压A 初始化中
ANDNOT D1052.04  ; 4St_1热压A 联锁
OUT D1050.02  ; 4St_1热压A工站运行
; rung 4: 1.0原点位
LD D1055.00  ; 4St_1热压A递进启动
OUT D1051.00
; rung 5: 2.0初始化
@LD D1052.12  ; 4St_1热压A 初始化[T]
@OR D1002.12  ; 整机初始化[T]
OR D1052.01  ; 4St_1热压A 初始化中
AND D1000.01  ; 手动模式
ANDNOT T0103  ; 复位按钮延时
AND D1052.00  ; 4St_1热压A工站就绪
ANDNOT D1050.00  ; 4St_1热压A工站错误
ANDNOT T0054  ; 3St-B初始位延时
OUT D1052.01  ; 4St_1热压A 初始化中
AND D1051.00
TIM 0054 #1  ; 3St-B初始位延时
; rung 6: 2.1自动停止CMD
LD D1000.01  ; 手动模式
ANDNOT D1052.01  ; 4St_1热压A 初始化中
AND D1052.15  ; 4St_1热压A 任务停止[T]
AND H1.00  ; 工位步序初始（1启用）
MOVL(498) &1 D1055  ; 3ST_B进出料移栽自动步序

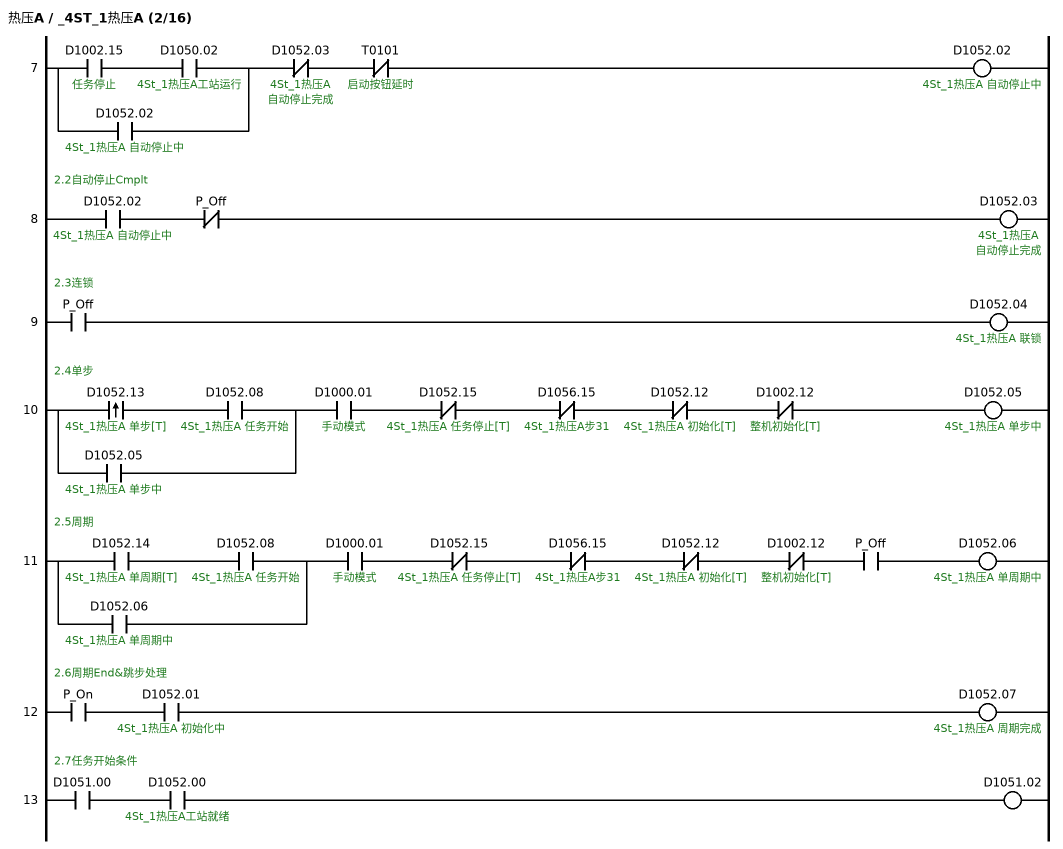
; rung 7
LD D1002.15  ; 任务停止
AND D1050.02  ; 4St_1热压A工站运行
OR D1052.02  ; 4St_1热压A 自动停止中
ANDNOT D1052.03  ; 4St_1热压A 自动停止完成
ANDNOT T0101  ; 启动按钮延时
OUT D1052.02  ; 4St_1热压A 自动停止中
; rung 8: 2.2自动停止Cmplt
LD D1052.02  ; 4St_1热压A 自动停止中
ANDNOT P_Off
OUT D1052.03  ; 4St_1热压A 自动停止完成
; rung 9: 2.3连锁
LD P_Off
OUT D1052.04  ; 4St_1热压A 联锁
; rung 10: 2.4单步
@LD D1052.13  ; 4St_1热压A 单步[T]
AND D1052.08  ; 4St_1热压A 任务开始
OR D1052.05  ; 4St_1热压A 单步中
AND D1000.01  ; 手动模式
ANDNOT D1052.15  ; 4St_1热压A 任务停止[T]
ANDNOT D1056.15  ; 4St_1热压A步31
ANDNOT D1052.12  ; 4St_1热压A 初始化[T]
ANDNOT D1002.12  ; 整机初始化[T]
OUT D1052.05  ; 4St_1热压A 单步中
; rung 11: 2.5周期
LD D1052.14  ; 4St_1热压A 单周期[T]
AND D1052.08  ; 4St_1热压A 任务开始
OR D1052.06  ; 4St_1热压A 单周期中
AND D1000.01  ; 手动模式
ANDNOT D1052.15  ; 4St_1热压A 任务停止[T]
ANDNOT D1056.15  ; 4St_1热压A步31
ANDNOT D1052.12  ; 4St_1热压A 初始化[T]
ANDNOT D1002.12  ; 整机初始化[T]
AND P_Off
OUT D1052.06  ; 4St_1热压A 单周期中
; rung 12: 2.6周期End&跳步处理
LD P_On
AND D1052.01  ; 4St_1热压A 初始化中
OUT D1052.07  ; 4St_1热压A 周期完成
; rung 13: 2.7任务开始条件
LD D1051.00
AND D1052.00  ; 4St_1热压A工站就绪
OUT D1051.02

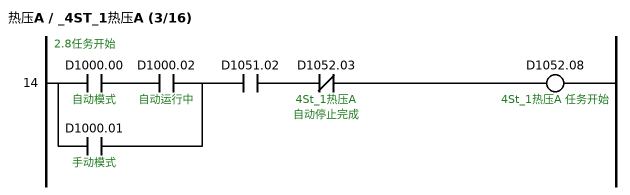
; rung 14: 2.8任务开始
LD D1000.00  ; 自动模式
AND D1000.02  ; 自动运行中
OR D1000.01  ; 手动模式
AND D1051.02
ANDNOT D1052.03  ; 4St_1热压A 自动停止完成
OUT D1052.08  ; 4St_1热压A 任务开始

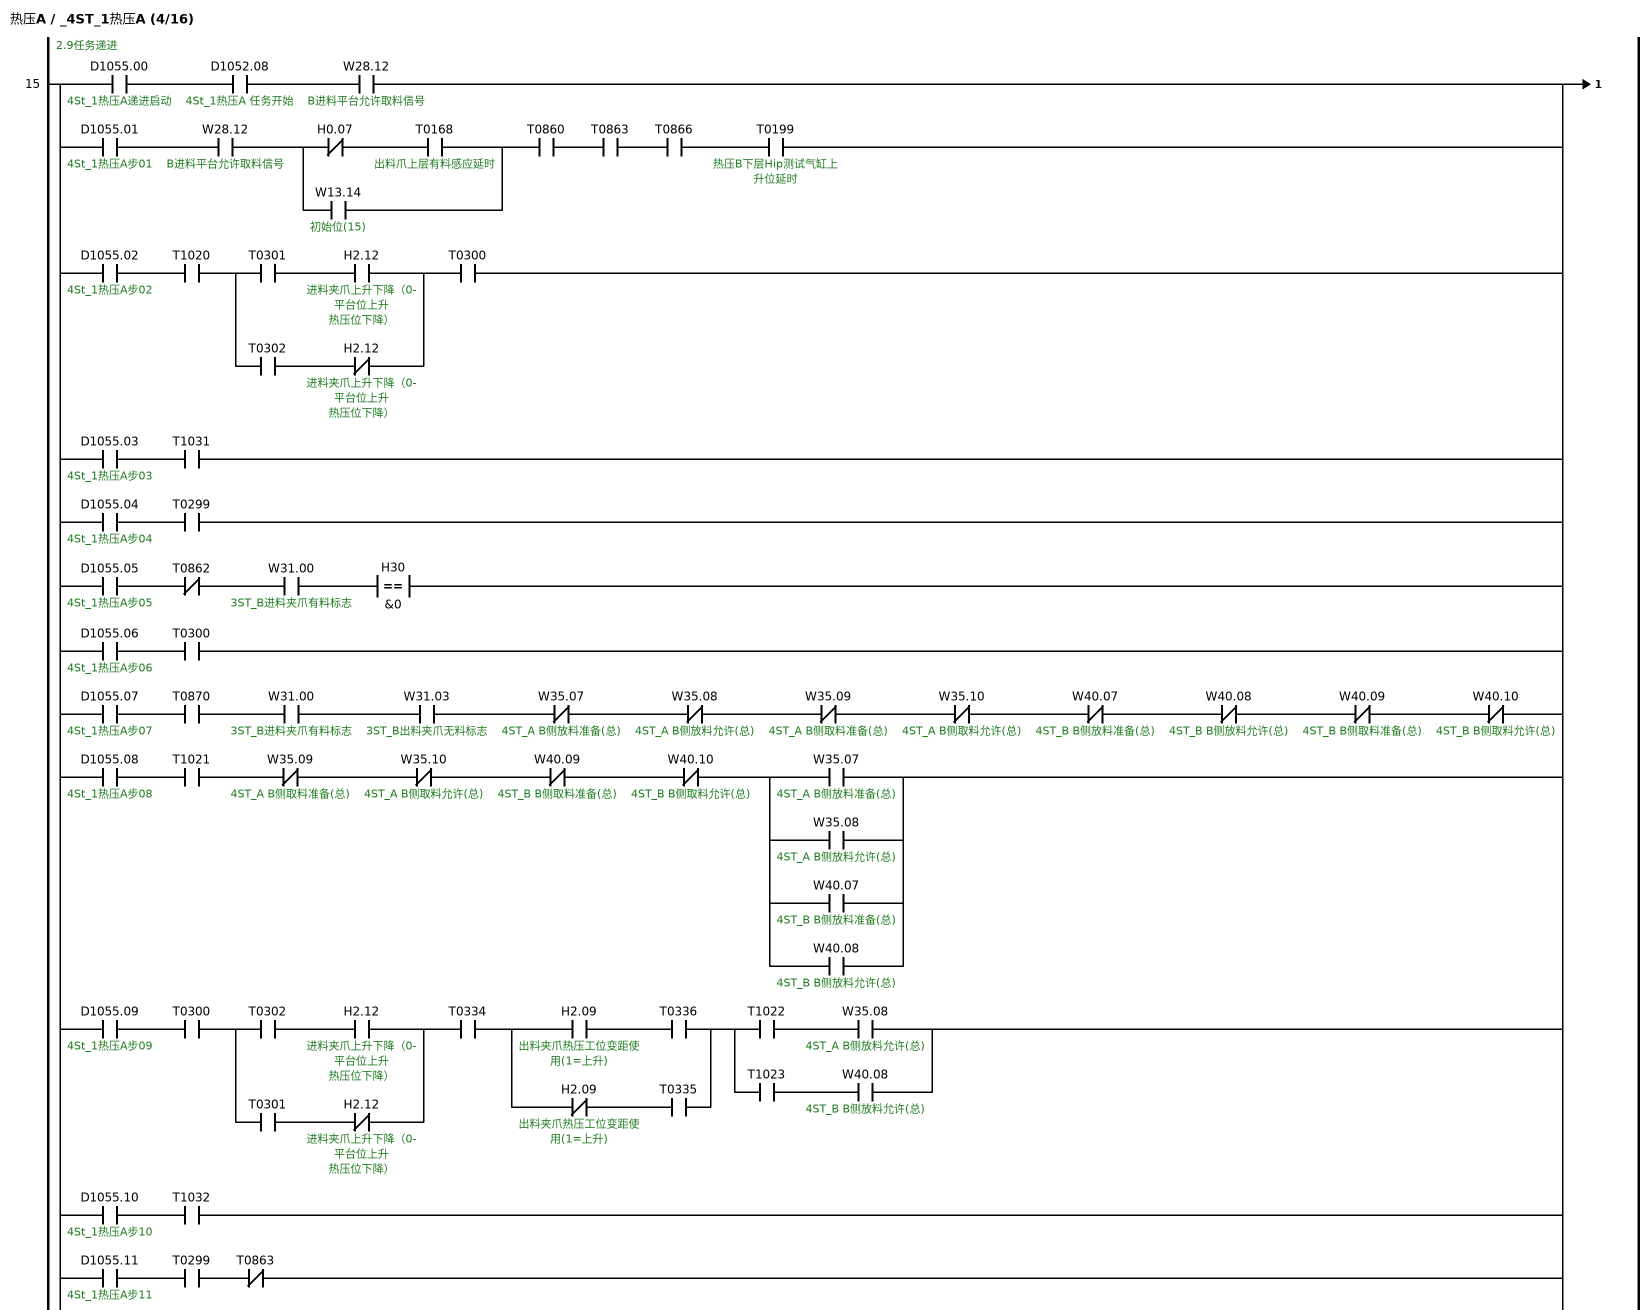

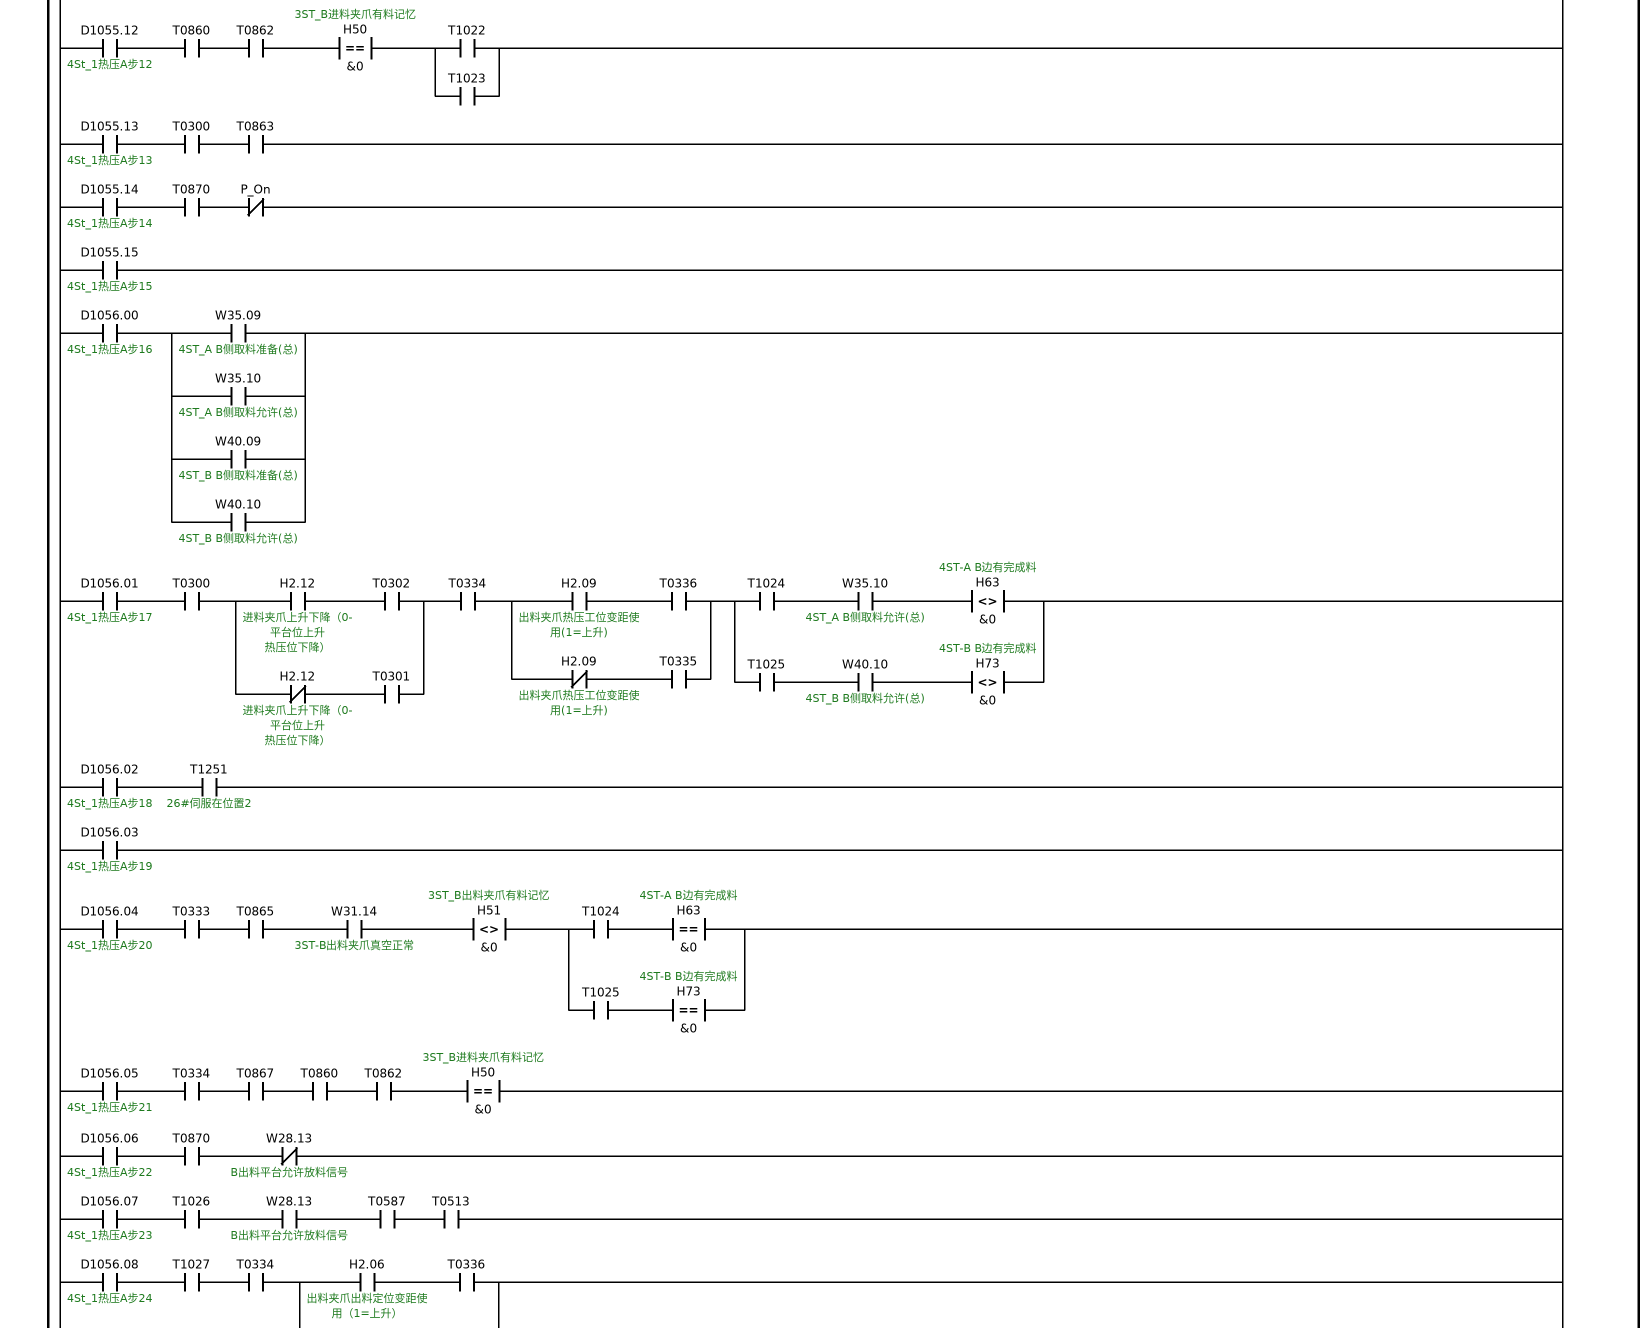

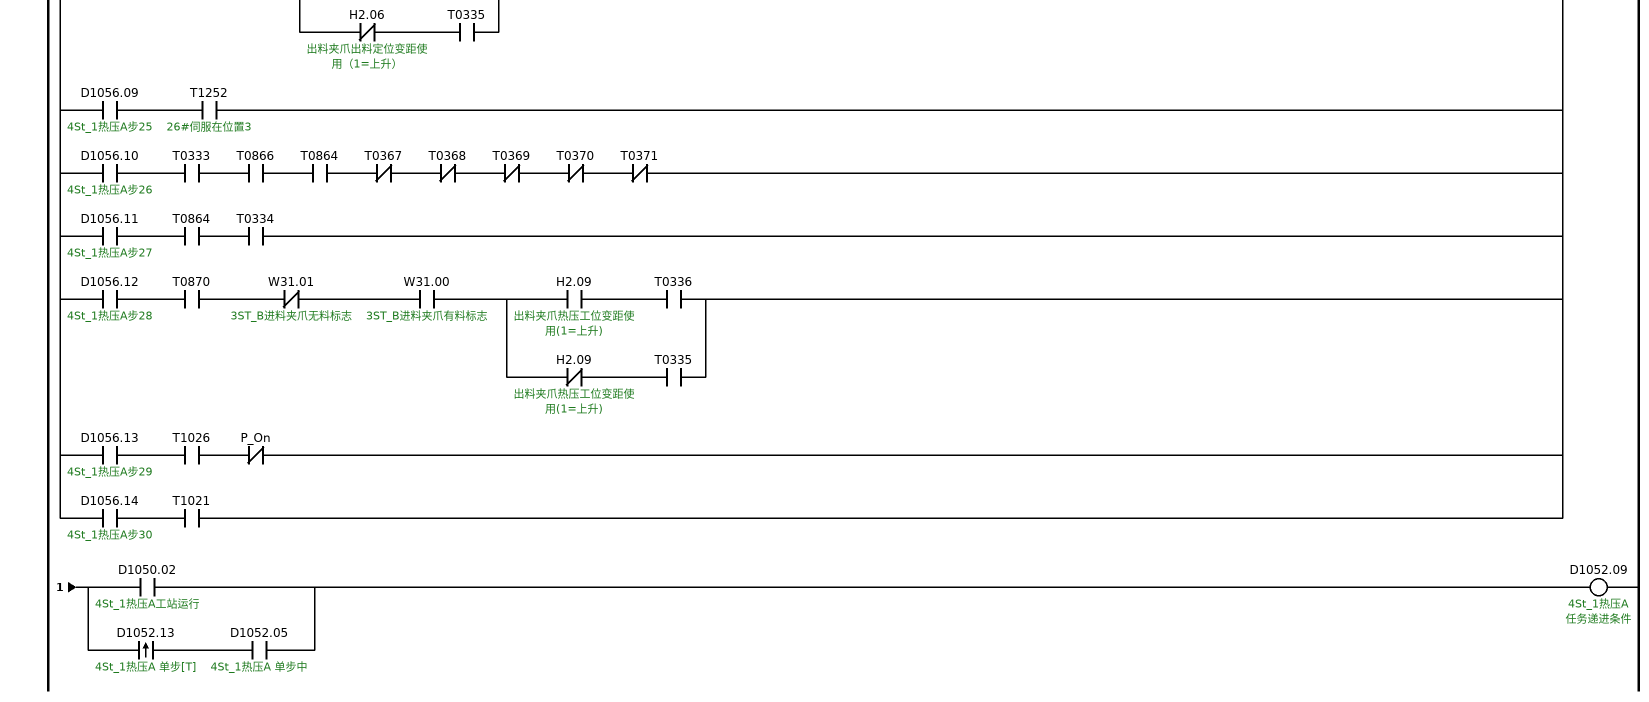
; rung 15: 2.9任务递进
LD D1055.00  ; 4St_1热压A递进启动
AND D1052.08  ; 4St_1热压A 任务开始
AND W28.12  ; B进料平台允许取料信号
LD D1055.01  ; 4St_1热压A步01
AND W28.12  ; B进料平台允许取料信号
LDNOT H0.07
AND T0168  ; 出料爪上层有料感应延时
OR W13.14  ; 初始位(15)
ANDLD
AND T0860
AND T0863
AND T0866
AND T0199  ; 热压B下层Hip测试气缸上升位延时
ORLD
LD D1055.02  ; 4St_1热压A步02
AND T1020
LD T0301
AND H2.12  ; 进料夹爪上升下降（0-平台位上升  热压位下降）
LD T0302
ANDNOT H2.12  ; 进料夹爪上升下降（0-平台位上升  热压位下降）
ORLD
ANDLD
AND T0300
ORLD
LD D1055.03  ; 4St_1热压A步03
AND T1031
ORLD
LD D1055.04  ; 4St_1热压A步04
AND T0299
ORLD
LD D1055.05  ; 4St_1热压A步05
ANDNOT T0862
AND W31.00  ; 3ST_B进料夹爪有料标志
AND=(300) H30 &0
ORLD
LD D1055.06  ; 4St_1热压A步06
AND T0300
ORLD
LD D1055.07  ; 4St_1热压A步07
AND T0870
AND W31.00  ; 3ST_B进料夹爪有料标志
AND W31.03  ; 3ST_B出料夹爪无料标志
ANDNOT W35.07  ; 4ST_A B侧放料准备(总)
ANDNOT W35.08  ; 4ST_A B侧放料允许(总)
ANDNOT W35.09  ; 4ST_A B侧取料准备(总)
ANDNOT W35.10  ; 4ST_A B侧取料允许(总)
ANDNOT W40.07  ; 4ST_B B侧放料准备(总)
ANDNOT W40.08  ; 4ST_B B侧放料允许(总)
ANDNOT W40.09  ; 4ST_B B侧取料准备(总)
ANDNOT W40.10  ; 4ST_B B侧取料允许(总)
ORLD
LD D1055.08  ; 4St_1热压A步08
AND T1021
ANDNOT W35.09  ; 4ST_A B侧取料准备(总)
ANDNOT W35.10  ; 4ST_A B侧取料允许(总)
ANDNOT W40.09  ; 4ST_B B侧取料准备(总)
ANDNOT W40.10  ; 4ST_B B侧取料允许(总)
LD W35.07  ; 4ST_A B侧放料准备(总)
OR W35.08  ; 4ST_A B侧放料允许(总)
OR W40.07  ; 4ST_B B侧放料准备(总)
OR W40.08  ; 4ST_B B侧放料允许(总)
ANDLD
ORLD
LD D1055.09  ; 4St_1热压A步09
AND T0300
LD T0302
AND H2.12  ; 进料夹爪上升下降（0-平台位上升  热压位下降）
LD T0301
ANDNOT H2.12  ; 进料夹爪上升下降（0-平台位上升  热压位下降）
ORLD
ANDLD
AND T0334
LD H2.09  ; 出料夹爪热压工位变距使用(1=上升)
AND T0336
LDNOT H2.09  ; 出料夹爪热压工位变距使用(1=上升)
AND T0335
ORLD
ANDLD
LD T1022
AND W35.08  ; 4ST_A B侧放料允许(总)
LD T1023
AND W40.08  ; 4ST_B B侧放料允许(总)
ORLD
ANDLD
ORLD
LD D1055.10  ; 4St_1热压A步10
AND T1032
ORLD
LD D1055.11  ; 4St_1热压A步11
AND T0299
ANDNOT T0863
ORLD
LD D1055.12  ; 4St_1热压A步12
AND T0860
AND T0862
AND=(300) H50 &0  ; 3ST_B进料夹爪有料记忆
LD T1022
OR T1023
ANDLD
ORLD
LD D1055.13  ; 4St_1热压A步13
AND T0300
AND T0863
ORLD
LD D1055.14  ; 4St_1热压A步14
AND T0870
ANDNOT P_On
ORLD
OR D1055.15  ; 4St_1热压A步15
LD D1056.00  ; 4St_1热压A步16
LD W35.09  ; 4ST_A B侧取料准备(总)
OR W35.10  ; 4ST_A B侧取料允许(总)
OR W40.09  ; 4ST_B B侧取料准备(总)
OR W40.10  ; 4ST_B B侧取料允许(总)
ANDLD
ORLD
LD D1056.01  ; 4St_1热压A步17
AND T0300
LD H2.12  ; 进料夹爪上升下降（0-平台位上升  热压位下降）
AND T0302
LDNOT H2.12  ; 进料夹爪上升下降（0-平台位上升  热压位下降）
AND T0301
ORLD
ANDLD
AND T0334
LD H2.09  ; 出料夹爪热压工位变距使用(1=上升)
AND T0336
LDNOT H2.09  ; 出料夹爪热压工位变距使用(1=上升)
AND T0335
ORLD
ANDLD
LD T1024
AND W35.10  ; 4ST_A B侧取料允许(总)
AND<>(305) H63 &0  ; 4ST-A B边有完成料
LD T1025
AND W40.10  ; 4ST_B B侧取料允许(总)
AND<>(305) H73 &0  ; 4ST-B B边有完成料
ORLD
ANDLD
ORLD
LD D1056.02  ; 4St_1热压A步18
AND T1251  ; 26#伺服在位置2
ORLD
OR D1056.03  ; 4St_1热压A步19
LD D1056.04  ; 4St_1热压A步20
AND T0333
AND T0865
AND W31.14  ; 3ST-B出料夹爪真空正常
AND<>(305) H51 &0  ; 3ST_B出料夹爪有料记忆
LD T1024
AND=(300) H63 &0  ; 4ST-A B边有完成料
LD T1025
AND=(300) H73 &0  ; 4ST-B B边有完成料
ORLD
ANDLD
ORLD
LD D1056.05  ; 4St_1热压A步21
AND T0334
AND T0867
AND T0860
AND T0862
AND=(300) H50 &0  ; 3ST_B进料夹爪有料记忆
ORLD
LD D1056.06  ; 4St_1热压A步22
AND T0870
ANDNOT W28.13  ; B出料平台允许放料信号
ORLD
LD D1056.07  ; 4St_1热压A步23
AND T1026
AND W28.13  ; B出料平台允许放料信号
AND T0587
AND T0513
ORLD
LD D1056.08  ; 4St_1热压A步24
AND T1027
AND T0334
LD H2.06  ; 出料夹爪出料定位变距使用（1=上升）
AND T0336
LDNOT H2.06  ; 出料夹爪出料定位变距使用（1=上升）
AND T0335
ORLD
ANDLD
ORLD
LD D1056.09  ; 4St_1热压A步25
AND T1252  ; 26#伺服在位置3
ORLD
LD D1056.10  ; 4St_1热压A步26
AND T0333
AND T0866
AND T0864
ANDNOT T0367
ANDNOT T0368
ANDNOT T0369
ANDNOT T0370
ANDNOT T0371
ORLD
LD D1056.11  ; 4St_1热压A步27
AND T0864
AND T0334
ORLD
LD D1056.12  ; 4St_1热压A步28
AND T0870
ANDNOT W31.01  ; 3ST_B进料夹爪无料标志
AND W31.00  ; 3ST_B进料夹爪有料标志
LD H2.09  ; 出料夹爪热压工位变距使用(1=上升)
AND T0336
LDNOT H2.09  ; 出料夹爪热压工位变距使用(1=上升)
AND T0335
ORLD
ANDLD
ORLD
LD D1056.13  ; 4St_1热压A步29
AND T1026
ANDNOT P_On
ORLD
LD D1056.14  ; 4St_1热压A步30
AND T1021
ORLD
LD D1050.02  ; 4St_1热压A工站运行
@LD D1052.13  ; 4St_1热压A 单步[T]
AND D1052.05  ; 4St_1热压A 单步中
ORLD
ANDLD
OUT D1052.09  ; 4St_1热压A 任务递进条件

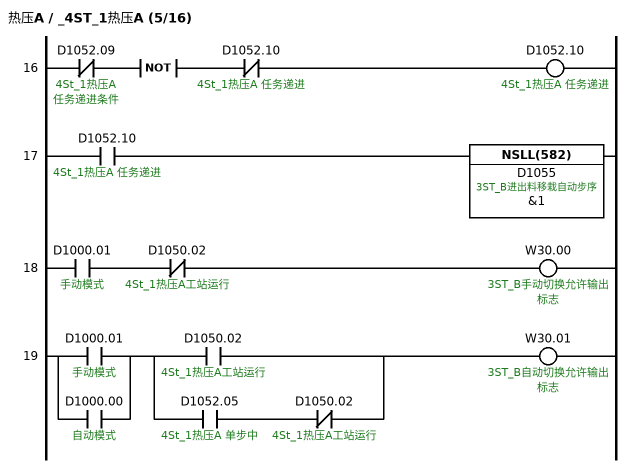
; rung 16
LDNOT D1052.09  ; 4St_1热压A 任务递进条件
NOT(520)
ANDNOT D1052.10  ; 4St_1热压A 任务递进
OUT D1052.10  ; 4St_1热压A 任务递进
; rung 17
LD D1052.10  ; 4St_1热压A 任务递进
NSLL(582) D1055 &1  ; 3ST_B进出料移栽自动步序
; rung 18
LD D1000.01  ; 手动模式
ANDNOT D1050.02  ; 4St_1热压A工站运行
OUT W30.00  ; 3ST_B手动切换允许输出标志
; rung 19
LD D1000.01  ; 手动模式
OR D1000.00  ; 自动模式
LD D1050.02  ; 4St_1热压A工站运行
LD D1052.05  ; 4St_1热压A 单步中
ANDNOT D1050.02  ; 4St_1热压A工站运行
ORLD
ANDLD
OUT W30.01  ; 3ST_B自动切换允许输出标志

